// Se o sinal não mudou de estado...
IF bPulse_2s = Special_Variables.Pulse_2s THEN
	// Atualiza temporizador do sinal
	di2sTimer:= di2sTimer + ProjectConstants.iMainTaskInterval;
	// Indica erro caso o sinal não tenha mudado de estado no dobro do tempo esperado
	IF di2sTimer > 2000 THEN bPulse2sFail:= TRUE; END_IF
// Se o sinal mudou de estado...
ELSE
	// Indica erro caso o sinal tenha mudado de estado antes ou depois do tempo esperado
	IF	di2sTimer < (2000 / 2 - diMainTaskIntervalGapMs) OR
		di2sTimer > (2000 / 2 + diMainTaskIntervalGapMs) THEN
			bPulse2sFail:= TRUE;
	END_IF
	// Inicializa o temporizador do sinal
	di2sTimer:= ProjectConstants.iMainTaskInterval;
	// Memoriza o estado atual do sinal
	bPulse_2s:= Special_Variables.Pulse_2s;
END_IF

// Se o sinal não mudou de estado...
IF bPulse_5s = Special_Variables.Pulse_5s THEN
	// Atualiza temporizador do sinal
	di5sTimer:= di5sTimer + ProjectConstants.iMainTaskInterval;
	// Indica erro caso o sinal não tenha mudado de estado no dobro do tempo esperado
	IF di5sTimer > 5000 THEN bPulse5sFail:= TRUE; END_IF
// Se o sinal mudou de estado...
ELSE
	// Indica erro caso o sinal tenha mudado de estado antes ou depois do tempo esperado
	IF	di5sTimer < (5000 / 2 - diMainTaskIntervalGapMs) OR
		di5sTimer > (5000 / 2 + diMainTaskIntervalGapMs) THEN
			bPulse5sFail:= TRUE;
	END_IF
	// Inicializa o temporizador do sinal
	di5sTimer:= ProjectConstants.iMainTaskInterval;
	// Memoriza o estado atual do sinal
	bPulse_5s:= Special_Variables.Pulse_5s;
END_IF

// Se o sinal não mudou de estado...
IF bPulse_10s = Special_Variables.Pulse_10s THEN
	// Atualiza temporizador do sinal
	di10sTimer:= di10sTimer + ProjectConstants.iMainTaskInterval;
	// Indica erro caso o sinal não tenha mudado de estado no dobro do tempo esperado
	IF di10sTimer > 10000 THEN bPulse10sFail:= TRUE; END_IF
// Se o sinal mudou de estado...
ELSE
	// Indica erro caso o sinal tenha mudado de estado antes ou depois do tempo esperado
	IF	di10sTimer < (10000 / 2 - diMainTaskIntervalGapMs) OR
		di10sTimer > (10000 / 2 + diMainTaskIntervalGapMs) THEN
			bPulse10sFail:= TRUE;
	END_IF
	// Inicializa o temporizador do sinal
	di10sTimer:= ProjectConstants.iMainTaskInterval;
	// Memoriza o estado atual do sinal
	bPulse_10s:= Special_Variables.Pulse_10s;
END_IF

// Se o sinal não mudou de estado...
IF bPulse_30s = Special_Variables.Pulse_30s THEN
	// Atualiza temporizador do sinal
	di30sTimer:= di30sTimer + ProjectConstants.iMainTaskInterval;
	// Indica erro caso o sinal não tenha mudado de estado no dobro do tempo esperado
	IF di30sTimer > 30000 THEN bPulse30sFail:= TRUE; END_IF
// Se o sinal mudou de estado...
ELSE
	// Indica erro caso o sinal tenha mudado de estado antes ou depois do tempo esperado
	IF	di30sTimer < (30000 / 2 - diMainTaskIntervalGapMs) OR
		di30sTimer > (30000 / 2 + diMainTaskIntervalGapMs) THEN
			bPulse30sFail:= TRUE;
	END_IF
	// Inicializa o temporizador do sinal
	di30sTimer:= ProjectConstants.iMainTaskInterval;
	// Memoriza o estado atual do sinal
	bPulse_30s:= Special_Variables.Pulse_30s;
END_IF

// Se o sinal não mudou de estado...
IF bPulse_60s = Special_Variables.Pulse_60s THEN
	// Atualiza temporizador do sinal
	di60sTimer:= di60sTimer + ProjectConstants.iMainTaskInterval;
	// Indica erro caso o sinal não tenha mudado de estado no dobro do tempo esperado
	IF di60sTimer > 60000 THEN bPulse60sFail:= TRUE; END_IF
// Se o sinal mudou de estado...
ELSE
	// Indica erro caso o sinal tenha mudado de estado antes ou depois do tempo esperado
	IF	di60sTimer < (60000 / 2 - diMainTaskIntervalGapMs) OR
		di60sTimer > (60000 / 2 + diMainTaskIntervalGapMs) THEN
			bPulse60sFail:= TRUE;
	END_IF
	// Inicializa o temporizador do sinal
	di60sTimer:= ProjectConstants.iMainTaskInterval;
	// Memoriza o estado atual do sinal
	bPulse_60s:= Special_Variables.Pulse_60s;
END_IF

// Realiza as consistências para identificar falhas nos demais sinais da GVL Special_Variables
bPulseScanFail:= bPulseScanFail OR Special_Variables.Pulse_Scan <> bPulse_Scan;
// Consistência em função do retorno da chamada da função
IF udiSystemTimeCall = NextoStandard.RTC_STATUS.NO_ERROR THEN
	// Só consiste se os milisegundos ainda não viraram...
	IF Special_Variables.System_Time.wMilliseconds <= System_Time.wMilliseconds THEN
		bSystemTimeFail:= bSystemTimeFail OR	Special_Variables.System_Time.byDayOfMonth <> System_Time.byDayOfMonth OR
												Special_Variables.System_Time.byHours <> System_Time.byHours OR
												Special_Variables.System_Time.byMinutes <> System_Time.byMinutes OR
												Special_Variables.System_Time.byMonth <> System_Time.byMonth OR
												Special_Variables.System_Time.bySeconds <> System_Time.bySeconds OR
												Special_Variables.System_Time.wYear <> System_Time.wYear;
		bHourMinuteFail:= bHourMinuteFail OR Special_Variables.Hour_Minute <> Hour_Minute;
		bDayOfWeekFail:= bDayOfWeekFail OR Special_Variables.Day_Of_Week <> Day_Of_Week;
	END_IF
ELSE
	// Indica que chamada de função retornou erro
	bSystemTimeCall:= TRUE;
	// Memoriza o erro para fins de depuração
	udiSystemTimeCallErr:= udiSystemTimeCall;
END_IF
bDayOfWeekNull:= bDayOfWeekNull OR Day_Of_Week = NextoStandard.DAYS_OF_WEEK.INVALID_DAY;
bMainTaskFail:= bMainTaskFail OR Special_Variables.udiMainTaskInterval <> DINT_TO_UDINT(ProjectConstants.iMainTaskInterval * 1000);

// Só consiste as variáveis especiais redundantes na UCP ativa, pois na UCP não-ativa elas estão um ciclo atrasadas
IF DG_NX4010.tRedundancy.RedDgnLoc.sGeneral_Diag.eRedState = REDUNDANCY_STATE.ACTIVE THEN
	// Realiza as consitências em relação as variáveis especiais redundantes
	CheckSpecialVarsRed();
END_IF

// Resume as falhas identificadas neste cluster
NonRedPointer.pbSpecialVariablesLoc^:=	bPulse100msFail	OR	CheckSpecialVarsRed.bPulse100msFail OR
										bPulse500msFail OR	CheckSpecialVarsRed.bPulse500msFail OR
										bPulse1sFail	OR	CheckSpecialVarsRed.bPulse1sFail OR
										bPulse2sFail	OR	CheckSpecialVarsRed.bPulse2sFail OR
										bPulse5sFail	OR	CheckSpecialVarsRed.bPulse5sFail OR
										bPulse10sFail	OR	CheckSpecialVarsRed.bPulse10sFail OR
										bPulse30sFail	OR	CheckSpecialVarsRed.bPulse30sFail OR
										bPulse60sFail	OR	CheckSpecialVarsRed.bPulse60sFail OR
										bPulseScanFail	OR	CheckSpecialVarsRed.bPulseScanFail OR
										bSystemTimeCall	OR
										bSystemTimeFail	OR
										bHourMinuteFail	OR
										bDayOfWeekFail	OR
										bDayOfWeekNull	OR
										bMainTaskFail	OR
										FALSE;

// Resume as falhas identificadas em ambos os clusters
PersistentVars.bSpecialVariables:=	PersistentVars.bSpecialVariables OR
									NonRedPointer.pbSpecialVariablesLoc^ OR
									NonRedPointer.pbSpecialVariablesRem^ OR
									FALSE;

// Registra o tempo do sistema
Return_SysTimeGetUs_2:= SysTimeCore.SysTimeGetUs(uliPouEndTime);

// Calcula duração mínima/máxima desta POU
MinMaxTimes.uliPouMinTime_CheckSpecialVars:= MIN(MinMaxTimes.uliPouMinTime_CheckSpecialVars, uliPouEndTime - uliPouIniTime);
MinMaxTimes.uliPouMaxTime_CheckSpecialVars:= MAX(MinMaxTimes.uliPouMaxTime_CheckSpecialVars, uliPouEndTime - uliPouIniTime);

END_PROGRAM

// Device/Application/UserPOUs/NonSkippedPrg
PROGRAM NonSkippedPrg
VAR
	{attribute 'symbol' := 'read'}
	OPCRedundancyActive : BOOL;
	byLocalRedStateOld : REDUNDANCY_STATE;
	uliPouIniTime : ULINT;
	uliPouEndTime : ULINT;
	uliPouAvgTime : ARRAY [1..100] OF ULINT;
	uliPouSumTime : ULINT;
	iPouTimeIndex : INT := 1;
	bFirstCycle : BOOL := 1;
	iIndex : INT;
	tonNetVar : TON;
	tTimeNetVar : TIME := TIME#2S0MS;
	
	udiContadorDeCallBack_Last : UDINT;
	udiContadorDeCallBack_timeout : UDINT;
	udiContadorDeCallBack_timeout_max : UDINT;
		
	{attribute 'symbol' := 'read'}
	DG_NX3030_ACTIVE_tDetailed_Thermometer_diTemperature : DINT;	
	
END_VAR

// Registra o tempo do sistema
SysTimeGetUs(uliPouIniTime);

// Registra a data e hora desta chamada (utilizado em várias POUs)
NextoStandard.GetDateAndTime(NonRedData.xNonSkippedPrgDateAndTime);

// Consistência das variáveis especiais (chamada cíclica)
CheckSpecialVariables();

tonNetVar.PT:=tTimeNetVar;
// Código utilizado na redundância OPC
IF fbRedundancyManagement.m_fbDiagnosticsLocal.eRedState = REDUNDANCY_STATE.ACTIVE THEN
      OPCRedundancyActive := TRUE;
	  tonNetVar();
	  tonNetVar.IN:=TRUE;
	  IF tonNetVar.Q = TRUE THEN
		  NetVar_Application_GVL.TxPDOs_UDP[0].bActive:=TRUE;
		  NetVar_Application_GVL.TxPDOs_UDP[1].bActive:=TRUE;
		  NetVar_Application_GVL.TxPDOs_UDP[2].bActive:=TRUE;
		  NetVar_Application_GVL.TxPDOs_UDP[3].bActive:=TRUE;
		  NetVar_Application_GVL.TxPDOs_UDP[4].bActive:=TRUE;
	  END_IF
ELSE
      OPCRedundancyActive := FALSE;
	  NetVar_Application_GVL.TxPDOs_UDP[0].bActive:=FALSE;
	  NetVar_Application_GVL.TxPDOs_UDP[1].bActive:=FALSE;
	  NetVar_Application_GVL.TxPDOs_UDP[2].bActive:=FALSE;
	  NetVar_Application_GVL.TxPDOs_UDP[3].bActive:=FALSE;
	  NetVar_Application_GVL.TxPDOs_UDP[4].bActive:=FALSE;
	  tonNetVar.IN:=FALSE;
END_IF

// Rotina responsável pela leitura das informações de firmware dos módulos do barramento local
IF DG_NX3030.tSummarized.bAbsentModules <> 0 OR SymbolicsNonRedundant.bReadHWVersions = FALSE THEN
	// Realiza Leitura do FW dos módulos no barramento
	ReadHwVersions();
END_IF
// Rotina que envia as informações de firmware do cluster não ativo para o ativo
WriteHwVersionsNonActive();

// Rotina de salvamento do estado de redundância deste PLC dos ciclos anteriores
NonRedData.aeLastRedState[2]:= NonRedData.aeLastRedState[1];
NonRedData.aeLastRedState[1]:= NonRedData.aeLastRedState[0];
NonRedData.aeLastRedState[0]:= DG_NX4010.tRedundancy.RedDgnLoc.sGeneral_Diag.eRedState;

// MODBUS_Slave_1: copia o valor das saídas para as entradas
ATs.abyModbus1Status:= ATs.abyModbus1Coils;
ATs.awModbus1InputReg:= ATs.awModbus1Holding;

// Comunicação MQTT
IF fbRedundancyManagement.m_fbDiagnosticsLocal.eRedState = REDUNDANCY_STATE.ACTIVE THEN
	MQTT();
END_IF


DG_NX3030_ACTIVE_tDetailed_Thermometer_diTemperature:= DG_NX3030.tDetailed.Thermometer.diTemperature;


// Faz uma copia do pedido de inicio do teste para uso nas demais POUs
Symbolics.bStartTestCopy:= PersistentVars.bStartTest;
// Retorna se o teste estiver desabilitado
IF PersistentVars.bStartTest = FALSE THEN
	RETURN;
END_IF

// Verifica solicitação de reinicialização do super teste
IF PersistentVars.bEnableCleanStats = TRUE THEN
	// Reseta solicitação de reinicialização
	PersistentVars.bEnableCleanStats:= FALSE;
	// Solicita a incialização de todas as variáveis
	CleanStats();
	SymbolicsNonRedundant.bReadHWVersions:= FALSE;
	SymbolicsNonRedundant.bEnableCleanStats_CheckForcing:= TRUE;
	SymbolicsNonRedundant.bEnableCleanStats_CheckRam:= TRUE;
	SymbolicsNonRedundant.bEnableCleanStats_CheckSntp:= TRUE;
	SymbolicsNonRedundant.bEnableCleanStats_CheckRedData:= TRUE;
	Symbolics.bEnableCleanStats_ActivePrg:= TRUE;
	Symbolics.bEnableCleanStats_CheckNVL:= TRUE;
	SymbolicsNonRedundant.bEnableCleanStats_NonSkippedPrg:= TRUE;
	SymbolicsNonRedundant.bEnableCleanStats_CheckDiagsRetain:= TRUE;
END_IF


CycleTimes();			// Registra os tempos de ciclo máximo, mínimo e médio das tarefas
CheckModbus1();			// Consistência dos objetos de comunicação MODBUS Serial
CheckRedData();			// Consistência dos dados redundantes
CheckSntp();			// Consistência da atualização do relógio via SNTP
UserLog();				// Consistência e geração do LOG de usuário
CheckForcing();			// Consistência dos forçamentos
CheckDiagsRetain();		// Consistência e resumo dos diagnósticos ativos
CheckRam();				// Consistência da memória RAM da UCP	
//DaylightSavingTime();	// Ajuste do timezone em função do horário de verão

// Reseta a indicação de alteração de estado de redundância deste PLC
NonRedData.bRedStateChanged:= FALSE;
// Detecta alteração no estado de redundância deste PLC
IF DG_NX4010.tRedundancy.RedDgnLoc.sGeneral_Diag.eRedState <> byLocalRedStateOld THEN
	// Salva o estado de redundância atual deste PLC
	byLocalRedStateOld:= DG_NX4010.tRedundancy.RedDgnLoc.sGeneral_Diag.eRedState;
	// Indica que o estado de redundância deste PLC alterou
	NonRedData.bRedStateChanged:= TRUE;
	// Se este PLC é o ativo...
	IF DG_NX4010.tRedundancy.RedDgnLoc.sGeneral_Diag.eRedState = REDUNDANCY_STATE.ACTIVE THEN
		// Habilita os MODBUS Ethernet clientes 
		System_Diagnostics.DG_MODBUS_Client_2.tCommand.bRestart:= TRUE;
		System_Diagnostics.DG_MODBUS_Client_3.tCommand.bRestart:= TRUE;
		System_Diagnostics.DG_MODBUS_Client_4.tCommand.bRestart:= TRUE;
	// Se este PLC é não-ativo...
	ELSE
		// Desabilita os MODBUS Ethernet clientes
		System_Diagnostics.DG_MODBUS_Client_2.tCommand.bStop:= TRUE;
		System_Diagnostics.DG_MODBUS_Client_3.tCommand.bStop:= TRUE;
		System_Diagnostics.DG_MODBUS_Client_4.tCommand.bStop:= TRUE;
		// Inicializa temporizador para atrasar a consistência dos valores lidos,
		// pois quando o PLC irá assumir como ativo, vai levar alguns ciclos até
		// que a comunicação MODBUS/Profibus seja estabelecida e estabilizada
		NonRedData.iProfibus5DigTimer:= - ProjectConstants.iTimeToSkipAsActive;
		NonRedData.iProfibus10AnaTimer:= - ProjectConstants.iTimeToSkipAsActive;
		NonRedData.iProfibus3DigTimer:= - ProjectConstants.iTimeToSkipAsActive;
		NonRedData.iProfibus98DigTimer:= - ProjectConstants.iTimeToSkipAsActive;
		NonRedData.iProfibus99DigTimer:= - ProjectConstants.iTimeToSkipAsActive;
		NonRedData.iProfibus99Dig1005Timer:= - ProjectConstants.iTimeToSkipAsActive;
		NonRedData.iProfibusNXTimer:= - ProjectConstants.iTimeToSkipAsActive;
		NonRedData.iProfibus99AnaTimer:= - ProjectConstants.iTimeToSkipAsActive;
		// Indicador de necessidade de inicializar as variáveis de geração de SOE
		// a partir dos diagnósticos retentivos
		NonRedData.bSoeFirstCheckCycle:= TRUE;
	END_IF
END_IF



/// Depuração do BUG 19183
IF SymbolicsNonRedundant.bEnableCleanStats_NonSkippedPrg THEN
	// Reseta os contadores de sobra de timeout da sincronismo
	FOR iIndex:= 0 TO 99 DO
		MinMaxTimes.auliRedRemainTimeoutCounter[iIndex]:= 0;
	END_FOR
	// Modifica o timeout de redundancia original (que era 111)
	redundancy_time_values.g_dwRedundancyTimeout_ms:= 151;
	SymbolicsNonRedundant.bEnableCleanStats_NonSkippedPrg:= FALSE;
ELSIF redundancy_time_values.g_uiLastTimeout <= 99 THEN
	// Incrementa a variável que conta o número de vezes que sobrou o respectivo tempo de sincronismo (índice) 
	MinMaxTimes.auliRedRemainTimeoutCounter[redundancy_time_values.g_uiLastTimeout]:= MinMaxTimes.auliRedRemainTimeoutCounter[redundancy_time_values.g_uiLastTimeout] + 1;
END_IF

//################################################################################################################


// Devido a 3S ter alterado o funcionamento do vfInit sem a Altus saber,
// o funcionamento da sincronização de ponteiros da redundância foi afetada.
// Essa variável interna "Callback_vfInit_Counter" sempre deve ser incrementada
// caso pare de incrementar, significa que a redundância pode apresentar problemas
// na sincronização dos dados.

IF fbRedundancyManagement.m_fbDiagnosticsLocal.eRedState = REDUNDANCY_STATE.STANDBY THEN
	// Confere se o valor mudou de um ciclo para outro
	IF Callback_vfInit_Counter <> udiContadorDeCallBack_Last THEN	
		udiContadorDeCallBack_Last:= Callback_vfInit_Counter;
		udiContadorDeCallBack_timeout:=0;
	ELSE
		udiContadorDeCallBack_timeout:= udiContadorDeCallBack_timeout+1;
	END_IF
	udiContadorDeCallBack_timeout_max:=MAX(udiContadorDeCallBack_timeout_max, udiContadorDeCallBack_timeout);
	// Todos os testes exeutados até agora, o valor máximo registrado foi 1.
	IF udiContadorDeCallBack_timeout_max > 1 THEN
		PersistentVars.iSyncFailCallback_vfInit:= PersistentVars.iSyncFailCallback_vfInit+1;
	END_IF
END_IF


//Esse hotfix deve ser usado quando em versões 3.11 a 3.13.
(* hotfix para versão 3.11 a 3.13 *)
 //  {implicit on}	
//   Callback_vfInit(0);
//   {implicit off}
//################################################################################################################



// Registra o tempo do sistema
SysTimeGetUs(uliPouEndTime);

// Calcula duração média desta POU
uliPouSumTime:= uliPouSumTime - uliPouAvgTime[iPouTimeIndex];
uliPouAvgTime[iPouTimeIndex]:= uliPouEndTime - uliPouIniTime;
uliPouSumTime:= uliPouSumTime + uliPouAvgTime[iPouTimeIndex];
// Calcula duração mínima/média/máxima desta POU
MinMaxTimes.uliPouMinTime_NonSkippedPrg:= MIN(MinMaxTimes.uliPouMinTime_NonSkippedPrg, uliPouAvgTime[iPouTimeIndex]);
MinMaxTimes.uliPouAvgTime_NonSkippedPrg:= uliPouSumTime/(SIZEOF(uliPouAvgTime)/SIZEOF(uliPouAvgTime[1]));
MinMaxTimes.uliPouMaxTime_NonSkippedPrg:= MAX(MinMaxTimes.uliPouMaxTime_NonSkippedPrg, uliPouAvgTime[iPouTimeIndex]);
// Proximo indice para cálculo da duração média desta POU
iPouTimeIndex:= iPouTimeIndex + 1;
IF iPouTimeIndex > ULINT_TO_INT(SIZEOF(uliPouAvgTime)/SIZEOF(uliPouAvgTime[1])) THEN
	iPouTimeIndex:= 1;
END_IF

END_PROGRAM

// Device/Application/UserPOUs/Non-Redundant/ReadHwVersions
PROGRAM ReadHwVersions
VAR
	pSlave : POINTER TO NextoSlave;
	dwRevisionID : ARRAY [0..31] OF DWORD;
	uiAddress : ARRAY [0..31] OF UINT;
	dwProductID : ARRAY [0..31] OF DWORD;
	byIndex : BYTE;
	iIndex : INT;
END_VAR

//*****************************************************************************
// Autor(es): Roberto Martiny
// Descrição:
// Esta POU realiza a leitura do firmware via NextoBus e armazena as informações para serem lidas via SCADA.
//*****************************************************************************

IF DG_NX4010.tRedundancy.RedDgnLoc.sGeneral_Diag.ePLC_ID = CLUCONF_ID.PLC_A THEN
	// Realiza a leitura do firmware via NextoBus. 
			IF g_pFirstMaster <> 0 THEN
			pSlave := g_pFirstMaster^.FirstSlave;
			///pSlave := Configuration.FirstSlave;
			WHILE pSlave <> 0 DO
			   dwRevisionID[byIndex] := pSlave^.RevisionID; // Leitura da versão fo firmware.
			   uiAddress[byIndex] := pSlave^.PhysSlaveAddr; // Leitura do rack e slot.
			   dwProductID[byIndex] := pSlave^.ProductID; // Leitura do tipo do produto.
			   byIndex:=byIndex+1;
			   pSlave := pSlave^.NextInstance;
			END_WHILE
			END_IF
		byIndex:= 0;
		
		FOR iIndex:=0 TO 31 DO
		// Consulta Informações Rack 00 Slot 04
			IF uiAddress[iIndex] = 16#0004 THEN
				HwVersions.eR00S04_NX4010_PlcA.iIndex:= iIndex;
			END_IF
			HwVersions.eR00S04_NX4010_PlcA.dwFirmwareVersion:= DwRevisionID[HwVersions.eR00S04_NX4010_PlcA.iIndex];
			HwVersions.eR00S04_NX4010_PlcA.dwProductID:= DwProductID[HwVersions.eR00S04_NX4010_PlcA.iIndex];
			HwVersions.eR00S04_NX4010_PlcA.uiSlaveAddress:= uiAddress[HwVersions.eR00S04_NX4010_PlcA.iIndex];
			
		// Consulta Informações Rack 00 Slot 06
			IF uiAddress[iIndex] = 16#0006 THEN
				HwVersions.eR00S06_NX5001_PlcA.iIndex:= iIndex;
			END_IF
			HwVersions.eR00S06_NX5001_PlcA.dwFirmwareVersion:= DwRevisionID[HwVersions.eR00S06_NX5001_PlcA.iIndex];
			HwVersions.eR00S06_NX5001_PlcA.dwProductID:= DwProductID[HwVersions.eR00S06_NX5001_PlcA.iIndex];
			HwVersions.eR00S06_NX5001_PlcA.uiSlaveAddress:= uiAddress[HwVersions.eR00S06_NX5001_PlcA.iIndex];	
			
		// Consulta Informações Rack 00 Slot 08
			IF uiAddress[iIndex] = 16#0008 THEN
				HwVersions.eR00S08_NX5001_PlcA.iIndex:= iIndex;
			END_IF
			HwVersions.eR00S08_NX5001_PlcA.dwFirmwareVersion:= DwRevisionID[HwVersions.eR00S08_NX5001_PlcA.iIndex];
			HwVersions.eR00S08_NX5001_PlcA.dwProductID:= DwProductID[HwVersions.eR00S08_NX5001_PlcA.iIndex];
			HwVersions.eR00S08_NX5001_PlcA.uiSlaveAddress:= uiAddress[HwVersions.eR00S08_NX5001_PlcA.iIndex];
	
		// Consulta Informações Rack 00 Slot 10
			IF uiAddress[iIndex] = 16#000A THEN
				HwVersions.eR00S10_NX5000_PlcA.iIndex:= iIndex;
			END_IF
			HwVersions.eR00S10_NX5000_PlcA.dwFirmwareVersion:= DwRevisionID[HwVersions.eR00S10_NX5000_PlcA.iIndex];
			HwVersions.eR00S10_NX5000_PlcA.dwProductID:= DwProductID[HwVersions.eR00S10_NX5000_PlcA.iIndex];
			HwVersions.eR00S10_NX5000_PlcA.uiSlaveAddress:= uiAddress[HwVersions.eR00S10_NX5000_PlcA.iIndex];
	
		// Consulta Informações Rack 00 Slot 12
			IF uiAddress[iIndex] = 16#000C THEN
				HwVersions.eR00S12_NX5000_PlcA.iIndex:= iIndex;
			END_IF
			HwVersions.eR00S12_NX5000_PlcA.dwFirmwareVersion:= DwRevisionID[HwVersions.eR00S12_NX5000_PlcA.iIndex];
			HwVersions.eR00S12_NX5000_PlcA.dwProductID:= DwProductID[HwVersions.eR00S12_NX5000_PlcA.iIndex];
			HwVersions.eR00S12_NX5000_PlcA.uiSlaveAddress:= uiAddress[HwVersions.eR00S12_NX5000_PlcA.iIndex];
			
		// Consulta Informações Rack 00 Slot 16
			IF uiAddress[iIndex] = 16#0010 THEN
				HwVersions.eR00S16_NX5001_PlcA.iIndex:= iIndex;
			END_IF
			HwVersions.eR00S16_NX5001_PlcA.dwFirmwareVersion:= DwRevisionID[HwVersions.eR00S16_NX5001_PlcA.iIndex];
			HwVersions.eR00S16_NX5001_PlcA.dwProductID:= DwProductID[HwVersions.eR00S16_NX5001_PlcA.iIndex];
			HwVersions.eR00S16_NX5001_PlcA.uiSlaveAddress:= uiAddress[HwVersions.eR00S16_NX5001_PlcA.iIndex];	
			
		// Consulta Informações Rack 00 Slot 20
			IF uiAddress[iIndex] = 16#0014 THEN
				HwVersions.eR00S20_NX5000_PlcA.iIndex:= iIndex;
			END_IF
			HwVersions.eR00S20_NX5000_PlcA.dwFirmwareVersion:= DwRevisionID[HwVersions.eR00S20_NX5000_PlcA.iIndex];
			HwVersions.eR00S20_NX5000_PlcA.dwProductID:= DwProductID[HwVersions.eR00S20_NX5000_PlcA.iIndex];
			HwVersions.eR00S20_NX5000_PlcA.uiSlaveAddress:= uiAddress[HwVersions.eR00S20_NX5000_PlcA.iIndex];			
		END_FOR	
	
		HwVersions.eR00S02_NX3030_PlcA.abyBootloaderVersion[0]:= DG_NX3030.tDetailed.Target.abyBootloaderVersion[0];
		HwVersions.eR00S02_NX3030_PlcA.abyBootloaderVersion[1]:= DG_NX3030.tDetailed.Target.abyBootloaderVersion[1];
		HwVersions.eR00S02_NX3030_PlcA.abyBootloaderVersion[2]:= DG_NX3030.tDetailed.Target.abyBootloaderVersion[2];
		HwVersions.eR00S02_NX3030_PlcA.abyBootloaderVersion[3]:= DG_NX3030.tDetailed.Target.abyBootloaderVersion[3];
		HwVersions.eR00S02_NX3030_PlcA.abyCPUVersion[0]:= DG_NX3030.tDetailed.Target.abyCPUVersion[0];
		HwVersions.eR00S02_NX3030_PlcA.abyCPUVersion[1]:= DG_NX3030.tDetailed.Target.abyCPUVersion[1];
		HwVersions.eR00S02_NX3030_PlcA.abyCPUVersion[2]:= DG_NX3030.tDetailed.Target.abyCPUVersion[2];
		HwVersions.eR00S02_NX3030_PlcA.abyCPUVersion[3]:= DG_NX3030.tDetailed.Target.abyCPUVersion[3];
		HwVersions.eR00S02_NX3030_PlcA.abyProcAuxVersion[0] := DG_NX3030.tDetailed.Target.abyAuxprocVersion[0];
		HwVersions.eR00S02_NX3030_PlcA.abyProcAuxVersion[1] := DG_NX3030.tDetailed.Target.abyAuxprocVersion[1];
		HwVersions.eR00S02_NX3030_PlcA.abyProcAuxVersion[2] := DG_NX3030.tDetailed.Target.abyAuxprocVersion[2];
		HwVersions.eR00S02_NX3030_PlcA.abyProcAuxVersion[3] := DG_NX3030.tDetailed.Target.abyAuxprocVersion[3];
		HwVersions.eR00S02_NX3030_PlcA.dwCPUModel:= DG_NX3030.tDetailed.Target.dwCPUModel;	
		
		SymbolicsNonRedundant.bReadHWVersions:= TRUE;
END_IF

IF DG_NX4010.tRedundancy.RedDgnLoc.sGeneral_Diag.ePLC_ID = CLUCONF_ID.PLC_B THEN
	// Realiza a leitura do firmware via NextoBus. 
			IF g_pFirstMaster <> 0 THEN
			pSlave := g_pFirstMaster^.FirstSlave;
			WHILE pSlave <> 0 DO
			   dwRevisionID[byIndex] := pSlave^.RevisionID; // Leitura da versão fo firmware.
			   uiAddress[byIndex] := pSlave^.PhysSlaveAddr; // Leitura do rack e slot.
			   dwProductID[byIndex] := pSlave^.ProductID; // Leitura do tipo do produto.
			   byIndex:=byIndex+1;
			   pSlave := pSlave^.NextInstance;
			END_WHILE
		byIndex:= 0;
		END_IF
		FOR iIndex:=0 TO 31 DO
			// Consulta Informações Rack 00 Slot 04
			IF uiAddress[iIndex] = 16#0004 THEN
				HwVersions.eR00S04_NX4010_PlcB.iIndex:= iIndex;
			END_IF
			HwVersions.eR00S04_NX4010_PlcB.dwFirmwareVersion:= DwRevisionID[HwVersions.eR00S04_NX4010_PlcB.iIndex];
			HwVersions.eR00S04_NX4010_PlcB.dwProductID:= DwProductID[HwVersions.eR00S04_NX4010_PlcB.iIndex];
			HwVersions.eR00S04_NX4010_PlcB.uiSlaveAddress:= uiAddress[HwVersions.eR00S04_NX4010_PlcB.iIndex];
			
		// Consulta Informações Rack 00 Slot 06
			IF uiAddress[iIndex] = 16#0006 THEN
				HwVersions.eR00S06_NX5001_PlcB.iIndex:= iIndex;
			END_IF
			HwVersions.eR00S06_NX5001_PlcB.dwFirmwareVersion:= DwRevisionID[HwVersions.eR00S06_NX5001_PlcB.iIndex];
			HwVersions.eR00S06_NX5001_PlcB.dwProductID:= DwProductID[HwVersions.eR00S06_NX5001_PlcB.iIndex];
			HwVersions.eR00S06_NX5001_PlcB.uiSlaveAddress:= uiAddress[HwVersions.eR00S06_NX5001_PlcB.iIndex];	
			
		// Consulta Informações Rack 00 Slot 08
			IF uiAddress[iIndex] = 16#0008 THEN
				HwVersions.eR00S08_NX5001_PlcB.iIndex:= iIndex;
			END_IF
			HwVersions.eR00S08_NX5001_PlcB.dwFirmwareVersion:= DwRevisionID[HwVersions.eR00S08_NX5001_PlcB.iIndex];
			HwVersions.eR00S08_NX5001_PlcB.dwProductID:= DwProductID[HwVersions.eR00S08_NX5001_PlcB.iIndex];
			HwVersions.eR00S08_NX5001_PlcB.uiSlaveAddress:= uiAddress[HwVersions.eR00S08_NX5001_PlcB.iIndex];
	
		// Consulta Informações Rack 00 Slot 10
			IF uiAddress[iIndex] = 16#000A THEN
				HwVersions.eR00S10_NX5000_PlcB.iIndex:= iIndex;
			END_IF
			HwVersions.eR00S10_NX5000_PlcB.dwFirmwareVersion:= DwRevisionID[HwVersions.eR00S10_NX5000_PlcB.iIndex];
			HwVersions.eR00S10_NX5000_PlcB.dwProductID:= DwProductID[HwVersions.eR00S10_NX5000_PlcB.iIndex];
			HwVersions.eR00S10_NX5000_PlcB.uiSlaveAddress:= uiAddress[HwVersions.eR00S10_NX5000_PlcB.iIndex];
	
		// Consulta Informações Rack 00 Slot 12
			IF uiAddress[iIndex] = 16#000C THEN
				HwVersions.eR00S12_NX5000_PlcB.iIndex:= iIndex;
			END_IF
			HwVersions.eR00S12_NX5000_PlcB.dwFirmwareVersion:= DwRevisionID[HwVersions.eR00S12_NX5000_PlcB.iIndex];
			HwVersions.eR00S12_NX5000_PlcB.dwProductID:= DwProductID[HwVersions.eR00S12_NX5000_PlcB.iIndex];
			HwVersions.eR00S12_NX5000_PlcB.uiSlaveAddress:= uiAddress[HwVersions.eR00S12_NX5000_PlcB.iIndex];
			
		// Consulta Informações Rack 00 Slot 16
			IF uiAddress[iIndex] = 16#0010 THEN
				HwVersions.eR00S16_NX5001_PlcB.iIndex:= iIndex;
			END_IF
			HwVersions.eR00S16_NX5001_PlcB.dwFirmwareVersion:= DwRevisionID[HwVersions.eR00S16_NX5001_PlcB.iIndex];
			HwVersions.eR00S16_NX5001_PlcB.dwProductID:= DwProductID[HwVersions.eR00S16_NX5001_PlcB.iIndex];
			HwVersions.eR00S16_NX5001_PlcB.uiSlaveAddress:= uiAddress[HwVersions.eR00S16_NX5001_PlcB.iIndex];	
			
		// Consulta Informações Rack 00 Slot 20
			IF uiAddress[iIndex] = 16#0014 THEN
				HwVersions.eR00S20_NX5000_PlcB.iIndex:= iIndex;
			END_IF
			HwVersions.eR00S20_NX5000_PlcB.dwFirmwareVersion:= DwRevisionID[HwVersions.eR00S20_NX5000_PlcB.iIndex];
			HwVersions.eR00S20_NX5000_PlcB.dwProductID:= DwProductID[HwVersions.eR00S20_NX5000_PlcB.iIndex];
			HwVersions.eR00S20_NX5000_PlcB.uiSlaveAddress:= uiAddress[HwVersions.eR00S20_NX5000_PlcB.iIndex];			
		END_FOR	
	
		HwVersions.eR00S02_NX3030_PlcB.abyBootloaderVersion[0]:= DG_NX3030.tDetailed.Target.abyBootloaderVersion[0];
		HwVersions.eR00S02_NX3030_PlcB.abyBootloaderVersion[1]:= DG_NX3030.tDetailed.Target.abyBootloaderVersion[1];
		HwVersions.eR00S02_NX3030_PlcB.abyBootloaderVersion[2]:= DG_NX3030.tDetailed.Target.abyBootloaderVersion[2];
		HwVersions.eR00S02_NX3030_PlcB.abyBootloaderVersion[3]:= DG_NX3030.tDetailed.Target.abyBootloaderVersion[3];
		HwVersions.eR00S02_NX3030_PlcB.abyCPUVersion[0]:= DG_NX3030.tDetailed.Target.abyCPUVersion[0];
		HwVersions.eR00S02_NX3030_PlcB.abyCPUVersion[1]:= DG_NX3030.tDetailed.Target.abyCPUVersion[1];
		HwVersions.eR00S02_NX3030_PlcB.abyCPUVersion[2]:= DG_NX3030.tDetailed.Target.abyCPUVersion[2];
		HwVersions.eR00S02_NX3030_PlcB.abyCPUVersion[3]:= DG_NX3030.tDetailed.Target.abyCPUVersion[3];
		HwVersions.eR00S02_NX3030_PlcB.abyProcAuxVersion[0] := DG_NX3030.tDetailed.Target.abyAuxprocVersion[0];
		HwVersions.eR00S02_NX3030_PlcB.abyProcAuxVersion[1] := DG_NX3030.tDetailed.Target.abyAuxprocVersion[1];
		HwVersions.eR00S02_NX3030_PlcB.abyProcAuxVersion[2] := DG_NX3030.tDetailed.Target.abyAuxprocVersion[2];
		HwVersions.eR00S02_NX3030_PlcB.abyProcAuxVersion[3] := DG_NX3030.tDetailed.Target.abyAuxprocVersion[3];
		HwVersions.eR00S02_NX3030_PlcB.dwCPUModel:= DG_NX3030.tDetailed.Target.dwCPUModel;
		
		SymbolicsNonRedundant.bReadHWVersions:= TRUE;
END_IF

END_PROGRAM

// Device/Application/UserPOUs/Non-Redundant/WriteHwVersionsNonActive
PROGRAM WriteHwVersionsNonActive
VAR
	pSlave : POINTER TO NextoSlave;
	dwRevisionID : ARRAY [0..31] OF DWORD;
	uiAddress : ARRAY [0..31] OF UINT;
	dwProductID : ARRAY [0..31] OF DWORD;
	byIndex : BYTE;
	iIndex : INT;
	uliPouIniTime : ULINT;
	uliPouEndTime : ULINT;
END_VAR

//*****************************************************************************
// Autor(es): Jenifer Dal Magro
// Descrição:
// Esta POU envia as versões de Hardware do PLC não Ativo para o Ativo.
//*****************************************************************************
// Registra o tempo do sistema
SysTimeGetUs(uliPouIniTime);

IF DG_NX4010.tRedundancy.RedDgnLoc.sGeneral_Diag.ePLC_ID = CLUCONF_ID.PLC_A THEN
	IF DG_NX4010.tRedundancy.RedDgnLoc.sGeneral_Diag.eRedState = REDUNDANCY_STATE.ACTIVE THEN
		// Copia as versões de Hardware do PLC B não ativo para suas posições na GVL HwVersions
		// Firmware da CPU
		HwVersions.eR00S02_NX3030_PlcB.abyCPUVersion[0]	:=	DG_NX4010.tRedundancy.RedUsrRem.abyUser[1]	;
		HwVersions.eR00S02_NX3030_PlcB.abyCPUVersion[1]	:=	DG_NX4010.tRedundancy.RedUsrRem.abyUser[2]	;
		HwVersions.eR00S02_NX3030_PlcB.abyCPUVersion[2]	:=	DG_NX4010.tRedundancy.RedUsrRem.abyUser[3]	;
		HwVersions.eR00S02_NX3030_PlcB.abyCPUVersion[3]	:=	DG_NX4010.tRedundancy.RedUsrRem.abyUser[4]	;
		// Bootloader
		HwVersions.eR00S02_NX3030_PlcB.abyBootloaderVersion[0]	:=	DG_NX4010.tRedundancy.RedUsrRem.abyUser[5]	;
		HwVersions.eR00S02_NX3030_PlcB.abyBootloaderVersion[1]	:=	DG_NX4010.tRedundancy.RedUsrRem.abyUser[6]	;
		HwVersions.eR00S02_NX3030_PlcB.abyBootloaderVersion[2]	:=	DG_NX4010.tRedundancy.RedUsrRem.abyUser[7]	;
		HwVersions.eR00S02_NX3030_PlcB.abyBootloaderVersion[3]	:=	DG_NX4010.tRedundancy.RedUsrRem.abyUser[8]	;
		// Pocessador Auxiliar
		HwVersions.eR00S02_NX3030_PlcB.abyProcAuxVersion[0]	:=	DG_NX4010.tRedundancy.RedUsrRem.abyUser[9]	;
		HwVersions.eR00S02_NX3030_PlcB.abyProcAuxVersion[1]	:=	DG_NX4010.tRedundancy.RedUsrRem.abyUser[10]	;
		HwVersions.eR00S02_NX3030_PlcB.abyProcAuxVersion[2]	:=	DG_NX4010.tRedundancy.RedUsrRem.abyUser[11]	;
		HwVersions.eR00S02_NX3030_PlcB.abyProcAuxVersion[3]	:=	DG_NX4010.tRedundancy.RedUsrRem.abyUser[12]	;	
		// Modelo CPU				
		HwVersions.eR00S02_NX3030_PlcB.dwCPUModel			:=	NonRedPointer.pdw02CPUModelRedUsrRem^	;
		// NX4010				
		HwVersions.eR00S04_NX4010_PlcB.dwFirmwareVersion	:=	NonRedPointer.pdw04NX4010FWRedUsrRem^	;
		HwVersions.eR00S04_NX4010_PlcB.dwProductID			:=	NonRedPointer.pdw04NX4010HWRedUsrRem^	;
		// NX50001				
		HwVersions.eR00S06_NX5001_PlcB.dwFirmwareVersion	:=	NonRedPointer.pdw06NX5001FWRedUsrRem^	;
		HwVersions.eR00S06_NX5001_PlcB.dwProductID			:=	NonRedPointer.pdw06NX5001HWRedUsrRem^	;
		HwVersions.eR00S08_NX5001_PlcB.dwFirmwareVersion	:=	NonRedPointer.pdw08NX5001FWRedUsrRem^	;
		HwVersions.eR00S08_NX5001_PlcB.dwProductID			:=	NonRedPointer.pdw08NX5001HWRedUsrRem^	;
		HwVersions.eR00S16_NX5001_PlcB.dwFirmwareVersion	:=	NonRedPointer.pdw16NX5001FWRedUsrRem^	;
		HwVersions.eR00S16_NX5001_PlcB.dwProductID			:=	NonRedPointer.pdw16NX5001HWRedUsrRem^	;
		// NX5000				
		HwVersions.eR00S10_NX5000_PlcB.dwFirmwareVersion	:=	NonRedPointer.pdw10NX5000FWRedUsrRem^	;
		HwVersions.eR00S10_NX5000_PlcB.dwProductID			:=	NonRedPointer.pdw10NX5000HWRedUsrRem^	;
		HwVersions.eR00S12_NX5000_PlcB.dwFirmwareVersion	:=	NonRedPointer.pdw12NX5000FWRedUsrRem^	;
		HwVersions.eR00S12_NX5000_PlcB.dwProductID			:=	NonRedPointer.pdw12NX5000HWRedUsrRem^	;
		HwVersions.eR00S20_NX5000_PlcB.dwFirmwareVersion	:=	NonRedPointer.pdw20NX5000FWRedUsrRem^	;
		HwVersions.eR00S20_NX5000_PlcB.dwProductID			:=	NonRedPointer.pdw20NX5000HWRedUsrRem^	;

		
	ELSIF	DG_NX4010.tRedundancy.RedDgnLoc.sGeneral_Diag.eRedState = REDUNDANCY_STATE.STANDBY	OR
			DG_NX4010.tRedundancy.RedDgnLoc.sGeneral_Diag.eRedState = REDUNDANCY_STATE.INACTIVE	THEN
		// Copia os dados deste PLC para a área de usuário do PLC remoto			
		// Firmware da CPU
		DG_NX4010.tRedundancy.RedUsrLoc.abyUser[1]	:=	HwVersions.eR00S02_NX3030_PlcA.abyCPUVersion[0]	;
		DG_NX4010.tRedundancy.RedUsrLoc.abyUser[2]	:=	HwVersions.eR00S02_NX3030_PlcA.abyCPUVersion[1]	;
		DG_NX4010.tRedundancy.RedUsrLoc.abyUser[3]	:=	HwVersions.eR00S02_NX3030_PlcA.abyCPUVersion[2]	;
		DG_NX4010.tRedundancy.RedUsrLoc.abyUser[4]	:=	HwVersions.eR00S02_NX3030_PlcA.abyCPUVersion[3]	;
		// Bootloader
		DG_NX4010.tRedundancy.RedUsrLoc.abyUser[5]	:=	HwVersions.eR00S02_NX3030_PlcA.abyBootloaderVersion[0]	;
		DG_NX4010.tRedundancy.RedUsrLoc.abyUser[6]	:=	HwVersions.eR00S02_NX3030_PlcA.abyBootloaderVersion[1]	;
		DG_NX4010.tRedundancy.RedUsrLoc.abyUser[7]	:=	HwVersions.eR00S02_NX3030_PlcA.abyBootloaderVersion[2]	;
		DG_NX4010.tRedundancy.RedUsrLoc.abyUser[8]	:=	HwVersions.eR00S02_NX3030_PlcA.abyBootloaderVersion[3]	;
		// Pocessador Auxiliar
		DG_NX4010.tRedundancy.RedUsrLoc.abyUser[9]	:=	HwVersions.eR00S02_NX3030_PlcA.abyProcAuxVersion[0]	;
		DG_NX4010.tRedundancy.RedUsrLoc.abyUser[10]	:=	HwVersions.eR00S02_NX3030_PlcA.abyProcAuxVersion[1]	;
		DG_NX4010.tRedundancy.RedUsrLoc.abyUser[11]	:=	HwVersions.eR00S02_NX3030_PlcA.abyProcAuxVersion[2]	;
		DG_NX4010.tRedundancy.RedUsrLoc.abyUser[12]	:=	HwVersions.eR00S02_NX3030_PlcA.abyProcAuxVersion[3]	;
		// Modelo CPU
		NonRedPointer.pdw02CPUModelRedUsrLoc^	:=	HwVersions.eR00S02_NX3030_PlcA.dwCPUModel	;
		// NX4010
		NonRedPointer.pdw04NX4010FWRedUsrLoc^	:=	HwVersions.eR00S04_NX4010_PlcA.dwFirmwareVersion	;
		NonRedPointer.pdw04NX4010HWRedUsrLoc^	:=	HwVersions.eR00S04_NX4010_PlcA.dwProductID	;
		// NX50001
		NonRedPointer.pdw06NX5001FWRedUsrLoc^	:=	HwVersions.eR00S06_NX5001_PlcA.dwFirmwareVersion	;
		NonRedPointer.pdw06NX5001HWRedUsrLoc^	:=	HwVersions.eR00S06_NX5001_PlcA.dwProductID	;
		NonRedPointer.pdw08NX5001FWRedUsrLoc^	:=	HwVersions.eR00S08_NX5001_PlcA.dwFirmwareVersion	;
		NonRedPointer.pdw08NX5001HWRedUsrLoc^	:=	HwVersions.eR00S08_NX5001_PlcA.dwProductID	;
		NonRedPointer.pdw16NX5001FWRedUsrLoc^	:=	HwVersions.eR00S16_NX5001_PlcA.dwFirmwareVersion	;
		NonRedPointer.pdw16NX5001HWRedUsrLoc^	:=	HwVersions.eR00S16_NX5001_PlcA.dwProductID	;
		// NX5000
		NonRedPointer.pdw10NX5000FWRedUsrLoc^	:=	HwVersions.eR00S10_NX5000_PlcA.dwFirmwareVersion	;
		NonRedPointer.pdw10NX5000HWRedUsrLoc^	:=	HwVersions.eR00S10_NX5000_PlcA.dwProductID	;
		NonRedPointer.pdw12NX5000FWRedUsrLoc^	:=	HwVersions.eR00S12_NX5000_PlcA.dwFirmwareVersion	;
		NonRedPointer.pdw12NX5000HWRedUsrLoc^	:=	HwVersions.eR00S12_NX5000_PlcA.dwProductID	;
		NonRedPointer.pdw20NX5000FWRedUsrLoc^	:=	HwVersions.eR00S20_NX5000_PlcA.dwFirmwareVersion	;
		NonRedPointer.pdw20NX5000HWRedUsrLoc^	:=	HwVersions.eR00S20_NX5000_PlcA.dwProductID	;

			
			
	END_IF
END_IF

IF DG_NX4010.tRedundancy.RedDgnLoc.sGeneral_Diag.ePLC_ID = CLUCONF_ID.PLC_B THEN
	IF DG_NX4010.tRedundancy.RedDgnLoc.sGeneral_Diag.eRedState = REDUNDANCY_STATE.ACTIVE THEN
		// Copia as versões de Hardware do PLC A não ativo para suas posições na GVL HwVersions
		// Firmware da CPU
		HwVersions.eR00S02_NX3030_PlcA.abyCPUVersion[0]	:=	DG_NX4010.tRedundancy.RedUsrRem.abyUser[1]	;
		HwVersions.eR00S02_NX3030_PlcA.abyCPUVersion[1]	:=	DG_NX4010.tRedundancy.RedUsrRem.abyUser[2]	;
		HwVersions.eR00S02_NX3030_PlcA.abyCPUVersion[2]	:=	DG_NX4010.tRedundancy.RedUsrRem.abyUser[3]	;
		HwVersions.eR00S02_NX3030_PlcA.abyCPUVersion[3]	:=	DG_NX4010.tRedundancy.RedUsrRem.abyUser[4]	;
		// Bootloader
		HwVersions.eR00S02_NX3030_PlcA.abyBootloaderVersion[0]	:=	DG_NX4010.tRedundancy.RedUsrRem.abyUser[5]	;
		HwVersions.eR00S02_NX3030_PlcA.abyBootloaderVersion[1]	:=	DG_NX4010.tRedundancy.RedUsrRem.abyUser[6]	;
		HwVersions.eR00S02_NX3030_PlcA.abyBootloaderVersion[2]	:=	DG_NX4010.tRedundancy.RedUsrRem.abyUser[7]	;
		HwVersions.eR00S02_NX3030_PlcA.abyBootloaderVersion[3]	:=	DG_NX4010.tRedundancy.RedUsrRem.abyUser[8]	;
		// Pocessador Auxiliar
		HwVersions.eR00S02_NX3030_PlcA.abyProcAuxVersion[0]	:=	DG_NX4010.tRedundancy.RedUsrRem.abyUser[9]	;
		HwVersions.eR00S02_NX3030_PlcA.abyProcAuxVersion[1]	:=	DG_NX4010.tRedundancy.RedUsrRem.abyUser[10]	;
		HwVersions.eR00S02_NX3030_PlcA.abyProcAuxVersion[2]	:=	DG_NX4010.tRedundancy.RedUsrRem.abyUser[11]	;
		HwVersions.eR00S02_NX3030_PlcA.abyProcAuxVersion[3]	:=	DG_NX4010.tRedundancy.RedUsrRem.abyUser[12]	;
		// Modelo CPU				
		HwVersions.eR00S02_NX3030_PlcA.dwCPUModel			:=	NonRedPointer.pdw02CPUModelRedUsrRem^	;
		// NX4010				
		HwVersions.eR00S04_NX4010_PlcA.dwFirmwareVersion	:=	NonRedPointer.pdw04NX4010FWRedUsrRem^	;
		HwVersions.eR00S04_NX4010_PlcA.dwProductID			:=	NonRedPointer.pdw04NX4010HWRedUsrRem^	;
		// NX50001				
		HwVersions.eR00S06_NX5001_PlcA.dwFirmwareVersion	:=	NonRedPointer.pdw06NX5001FWRedUsrRem^	;
		HwVersions.eR00S06_NX5001_PlcA.dwProductID			:=	NonRedPointer.pdw06NX5001HWRedUsrRem^	;
		HwVersions.eR00S08_NX5001_PlcA.dwFirmwareVersion	:=	NonRedPointer.pdw08NX5001FWRedUsrRem^	;
		HwVersions.eR00S08_NX5001_PlcA.dwProductID			:=	NonRedPointer.pdw08NX5001HWRedUsrRem^	;
		HwVersions.eR00S16_NX5001_PlcA.dwFirmwareVersion	:=	NonRedPointer.pdw16NX5001FWRedUsrRem^	;
		HwVersions.eR00S16_NX5001_PlcA.dwProductID			:=	NonRedPointer.pdw16NX5001HWRedUsrRem^	;
		// NX5000				
		HwVersions.eR00S10_NX5000_PlcA.dwFirmwareVersion	:=	NonRedPointer.pdw10NX5000FWRedUsrRem^	;
		HwVersions.eR00S10_NX5000_PlcA.dwProductID			:=	NonRedPointer.pdw10NX5000HWRedUsrRem^	;
		HwVersions.eR00S12_NX5000_PlcA.dwFirmwareVersion	:=	NonRedPointer.pdw12NX5000FWRedUsrRem^	;
		HwVersions.eR00S12_NX5000_PlcA.dwProductID			:=	NonRedPointer.pdw12NX5000HWRedUsrRem^	;
		HwVersions.eR00S20_NX5000_PlcA.dwFirmwareVersion	:=	NonRedPointer.pdw20NX5000FWRedUsrRem^	;
		HwVersions.eR00S20_NX5000_PlcA.dwProductID			:=	NonRedPointer.pdw20NX5000HWRedUsrRem^	;

	ELSIF	DG_NX4010.tRedundancy.RedDgnLoc.sGeneral_Diag.eRedState = REDUNDANCY_STATE.STANDBY	OR
			DG_NX4010.tRedundancy.RedDgnLoc.sGeneral_Diag.eRedState = REDUNDANCY_STATE.INACTIVE	THEN
		// Copia os dados deste PLC para a área de usuário do PLC remoto			
		// Firmware da CPU
		DG_NX4010.tRedundancy.RedUsrLoc.abyUser[1]	:=	HwVersions.eR00S02_NX3030_PlcB.abyCPUVersion[0]	;
		DG_NX4010.tRedundancy.RedUsrLoc.abyUser[2]	:=	HwVersions.eR00S02_NX3030_PlcB.abyCPUVersion[1]	;
		DG_NX4010.tRedundancy.RedUsrLoc.abyUser[3]	:=	HwVersions.eR00S02_NX3030_PlcB.abyCPUVersion[2]	;
		DG_NX4010.tRedundancy.RedUsrLoc.abyUser[4]	:=	HwVersions.eR00S02_NX3030_PlcB.abyCPUVersion[3]	;
		// Bootloader
		DG_NX4010.tRedundancy.RedUsrLoc.abyUser[5]	:=	HwVersions.eR00S02_NX3030_PlcB.abyBootloaderVersion[0]	;
		DG_NX4010.tRedundancy.RedUsrLoc.abyUser[6]	:=	HwVersions.eR00S02_NX3030_PlcB.abyBootloaderVersion[1]	;
		DG_NX4010.tRedundancy.RedUsrLoc.abyUser[7]	:=	HwVersions.eR00S02_NX3030_PlcB.abyBootloaderVersion[2]	;
		DG_NX4010.tRedundancy.RedUsrLoc.abyUser[8]	:=	HwVersions.eR00S02_NX3030_PlcB.abyBootloaderVersion[3]	;
		// Pocessador Auxiliar
		DG_NX4010.tRedundancy.RedUsrLoc.abyUser[9]	:=	HwVersions.eR00S02_NX3030_PlcB.abyProcAuxVersion[0]	;
		DG_NX4010.tRedundancy.RedUsrLoc.abyUser[10]	:=	HwVersions.eR00S02_NX3030_PlcB.abyProcAuxVersion[1]	;
		DG_NX4010.tRedundancy.RedUsrLoc.abyUser[11]	:=	HwVersions.eR00S02_NX3030_PlcB.abyProcAuxVersion[2]	;
		DG_NX4010.tRedundancy.RedUsrLoc.abyUser[12]	:=	HwVersions.eR00S02_NX3030_PlcB.abyProcAuxVersion[3]	;		
		// Modelo CPU
		NonRedPointer.pdw02CPUModelRedUsrLoc^	:=	HwVersions.eR00S02_NX3030_PlcB.dwCPUModel	;
		// NX4010
		NonRedPointer.pdw04NX4010FWRedUsrLoc^	:=	HwVersions.eR00S04_NX4010_PlcB.dwFirmwareVersion	;
		NonRedPointer.pdw04NX4010HWRedUsrLoc^	:=	HwVersions.eR00S04_NX4010_PlcB.dwProductID	;
		// NX50001
		NonRedPointer.pdw06NX5001FWRedUsrLoc^	:=	HwVersions.eR00S06_NX5001_PlcB.dwFirmwareVersion	;
		NonRedPointer.pdw06NX5001HWRedUsrLoc^	:=	HwVersions.eR00S06_NX5001_PlcB.dwProductID	;
		NonRedPointer.pdw08NX5001FWRedUsrLoc^	:=	HwVersions.eR00S08_NX5001_PlcB.dwFirmwareVersion	;
		NonRedPointer.pdw08NX5001HWRedUsrLoc^	:=	HwVersions.eR00S08_NX5001_PlcB.dwProductID	;
		NonRedPointer.pdw16NX5001FWRedUsrLoc^	:=	HwVersions.eR00S16_NX5001_PlcB.dwFirmwareVersion	;
		NonRedPointer.pdw16NX5001HWRedUsrLoc^	:=	HwVersions.eR00S16_NX5001_PlcB.dwProductID	;
		// NX5000
		NonRedPointer.pdw10NX5000FWRedUsrLoc^	:=	HwVersions.eR00S10_NX5000_PlcB.dwFirmwareVersion	;
		NonRedPointer.pdw10NX5000HWRedUsrLoc^	:=	HwVersions.eR00S10_NX5000_PlcB.dwProductID	;
		NonRedPointer.pdw12NX5000FWRedUsrLoc^	:=	HwVersions.eR00S12_NX5000_PlcB.dwFirmwareVersion	;
		NonRedPointer.pdw12NX5000HWRedUsrLoc^	:=	HwVersions.eR00S12_NX5000_PlcB.dwProductID	;
		NonRedPointer.pdw20NX5000FWRedUsrLoc^	:=	HwVersions.eR00S20_NX5000_PlcB.dwFirmwareVersion	;
		NonRedPointer.pdw20NX5000HWRedUsrLoc^	:=	HwVersions.eR00S20_NX5000_PlcB.dwProductID	;
		
	END_IF
END_IF

// Registra o tempo do sistema
SysTimeGetUs(uliPouEndTime);
// Calcula duração mínima/máxima desta POU
MinMaxTimes.uliPouMinTime_WriteHwVersionsNonActive:= MIN(MinMaxTimes.uliPouMinTime_WriteHwVersionsNonActive, uliPouEndTime - uliPouIniTime);
MinMaxTimes.uliPouMaxTime_WriteHwVersionsNonActive:= MAX(MinMaxTimes.uliPouMaxTime_WriteHwVersionsNonActive, uliPouEndTime - uliPouIniTime);

END_PROGRAM

// Device/Application/UserPOUs/Non-Redundant/MQTT
PROGRAM MQTT
VAR
// #######################################################################################	
	// Function Block -> Library LibMQTT	
	MQTT: LibMQTT.MQTT_CLIENT;
	CONN: LibMQTT.MQTT_CONN_CONFIG;
	SUBS: ARRAY [1..LibMQTT.gc_uiMaxSubs] OF LibMQTT.MQTT_SUBSCRIBE;
	PUBS: ARRAY [1..LibMQTT.gc_uiMaxPubs] OF LibMQTT.MQTT_PUBLISH;
	RCV: ARRAY [1..LibMQTT.gc_uiMaxSubs] OF LibMQTT.MQTT_RECEIVED;
	ENABLE: BOOL := TRUE; // Sempre vem habilitado o MQTT
	
	// Mensagem recebiba pelo subscriber
	sub1_RcvMessage : STRING;
	
	pub1_PubMessage : STRING;
	pub2_PubMessage : STRING;
	
	// Comando para disparar a publicação
	pub1_bEnablePublish : BOOL;
	pub2_bEnablePublish : BOOL;
	
	uliPouIniTime : ULINT;
	uliPouEndTime : ULINT;
END_VAR

// Registra o tempo do sistema
SysTimeGetUs(uliPouIniTime);

// Parâmetros de conexão com o Servidor A
CONN.bCleanSession :=TRUE;
CONN.sHostname := '192.168.16.86';
CONN.uiPort := 1883;       // Quando usado TLS porta deve ser 8883, caso contrário 1883.
CONN.uiKeepAlive := 60;
CONN.bEnableTLS := FALSE; // NX3010/20/30 não suportam TLS
CONN.sCertFilename := 'ca.crt';

// Parâmetros do Subscriber
SUBS[1].sSubscribeTopic := 'altus/jg03_NX3030/ElapsedTimeToFailure';
SUBS[1].eSubscribeQoS := LibMQTT.MQTT_QOS_2;
SUBS[1].pbPayloadBuffer := ADR(sub1_RcvMessage);
SUBS[1].uiMaxPayloadSize := SIZEOF(sub1_RcvMessage);

//Parâmetros do Publisher
PUBS[1].bEnablePublish := pub1_bEnablePublish AND NOT(MQTT.PUBLISH_STATUS[1]);
PUBS[1].sPublishTopic := 'altus/jg03_NX3030/ElapsedTimeToFailure';
PUBS[1].pbPublishPayload := ADR(pub1_PubMessage);
PUBS[1].uiPublishPayloadSize := INT_TO_UINT(LEN(pub1_PubMessage));
PUBS[1].ePublishMessageQoS := LibMQTT.MQTT_QOS_2;

//Parâmetros do Publisher
PUBS[2].bEnablePublish := pub2_bEnablePublish AND NOT(MQTT.PUBLISH_STATUS[2]);
PUBS[2].sPublishTopic := 'altus/jg03_NX3030/ElapsedTimeToFailureToScada';
PUBS[2].pbPublishPayload := ADR(pub2_PubMessage);
PUBS[2].uiPublishPayloadSize := INT_TO_UINT(LEN(pub2_PubMessage));
PUBS[2].ePublishMessageQoS := LibMQTT.MQTT_QOS_2;

// Chamada da função MQTT	
MQTT.ENABLE :=  (TRUE AND NOT(MQTT.ERROR));
MQTT.CONNECTION_CONFIG := CONN;
MQTT.SUBSCRIBE := SUBS;
MQTT.PUBLISH := PUBS;


// Somente chama a função se estiver no controlador correto.
// Essa consistência é devido ao pessoal do mtool utilizar projetos do superteste em outras CPUs.
IF (DG_NX3030.tDetailed.Ethernet.NET1.abyMAC[0] = 16#00 AND
	DG_NX3030.tDetailed.Ethernet.NET1.abyMAC[1] = 16#80 AND
	DG_NX3030.tDetailed.Ethernet.NET1.abyMAC[2] = 16#A0 AND
	DG_NX3030.tDetailed.Ethernet.NET1.abyMAC[3] = 16#05 AND
	DG_NX3030.tDetailed.Ethernet.NET1.abyMAC[4] = 16#F1 AND
	DG_NX3030.tDetailed.Ethernet.NET1.abyMAC[5] = 16#84) THEN
	MQTT();
END_IF


// Mensagem a ser publicada

// Para testar o MQTT por completo, uma mensagem é publicada no servidor,
// a mesma é lida pelo subscriber, e então enviado pelo segundo publisher que é mostrada na tela do SCADA
pub1_PubMessage := TIME_TO_STRING(PersistentVars.tElapsedTimeToFailure);
pub2_PubMessage:= sub1_RcvMessage;

// Dispara a publicação a cada 1 segundo, caso não tenha problemas de comunicação
IF MQTT.CONNECTED = TRUE AND 
	MQTT.STATE = LibMQTT.MQTT_STATES.MQTT_READY AND
	MQTT.ERROR = FALSE THEN
	
	pub1_bEnablePublish:= Special_Variables.Pulse_1s;
	pub2_bEnablePublish:= Special_Variables.Pulse_1s;
END_IF


// Registra o tempo do sistema
SysTimeGetUs(uliPouEndTime);
// Calcula duração mínima/máxima desta POU
MinMaxTimes.uliPouMinTime_MQTT:= MIN(MinMaxTimes.uliPouMinTime_MQTT, uliPouEndTime - uliPouIniTime);
MinMaxTimes.uliPouMaxTime_MQTT:= MAX(MinMaxTimes.uliPouMaxTime_MQTT, uliPouEndTime - uliPouIniTime);

END_PROGRAM

// Device/Application/UserPOUs/Non-Redundant/CleanStats
PROGRAM CleanStats
VAR
	uliPouIniTime : ULINT;
	uliPouEndTime : ULINT;
END_VAR
VAR RETAIN
	iCleanStatsCallCnt : INT := 0;
END_VAR

// POU que zera o relatório dos testes, que é retentivo.
// Precisa ser habilitada na ActivePrg.

// Registra o tempo do sistema
SysTimeGetUs(uliPouIniTime);

// Registra a chamada desta POU
iCleanStatsCallCnt:= iCleanStatsCallCnt + 1;

// Solicita reinicialização dos contadores do MODBUS
DG_MODBUS_Master_1.tCommand.bResetCounter:= TRUE;
DG_MODBUS_Slave_1.tCommand.bResetCounter:= TRUE;
DG_MODBUS_Client_2.tCommand.bResetCounter:= TRUE;
DG_MODBUS_Server_2.tCommand.bResetCounter:= TRUE;
DG_MODBUS_Client_3.tCommand.bResetCounter:= TRUE;
DG_MODBUS_Server_3.tCommand.bResetCounter:= TRUE;
DG_MODBUS_Client_4.tCommand.bResetCounter:= TRUE;
DG_MODBUS_Server_4.tCommand.bResetCounter:= TRUE;
// Solicita reinicialização dos contadores do NX4010
DG_NX4010.tRedundancy.RedCmdLoc.bResetNETStatisticsLocal:= TRUE;
DG_NX4010.tRedundancy.RedCmdLoc.bResetNETStatisticsRemote:= TRUE;
// Resultados da POU StateChange:
Persistentvars.bExchangeStateFail:= FALSE;
Persistentvars.dwTransitionsCnt:= 0;
Persistentvars.dwSwitchoverCnt:= 0;
// Resultados das POUs CheckRedData e IncrRedData:
Persistentvars.iSyncFailCntSymb:= 0;
Persistentvars.iSyncFailCntQ:= 0;
Persistentvars.iSyncFailCntM:= 0;
Persistentvars.iSyncFailCntI:= 0;
PersistentVars.iSyncFailCallback_vfInit :=0;
NonRedPointer.piSSyncFailLoc^:= 0;
NonRedPointer.piQSyncFailLoc^:= 0;
NonRedPointer.piMSyncFailLoc^:= 0;
NonRedPointer.piISyncFailLoc^:= 0;
NonRedPointer.piSSyncFailRem^:= 0;
NonRedPointer.piQSyncFailRem^:= 0;
NonRedPointer.piMSyncFailRem^:= 0;
NonRedPointer.piISyncFailRem^:= 0;
// Resultados da POU CycleTimes:
Symbolics.bPlcAMaxMinSetup:= TRUE;
Persistentvars.dwPLCAMainTaskLoadMax:= 0;	
Persistentvars.dwPLCAMainTaskLoadAvg:= 0;	
Persistentvars.dwPLCAMainTaskLoadMin:= 10000; 	
Symbolics.bPlcBMaxMinSetup:= TRUE;
Persistentvars.dwPLCBMainTaskLoadMax:= 0;
Persistentvars.dwPLCBMainTaskLoadAvg:= 0;	
Persistentvars.dwPLCBMainTaskLoadMin:= 10000;
// Resultados da POU CheckProfibusIOs:
Persistentvars.dwSlave5DigIOsErrors:= 0;
Persistentvars.dwSlave5Unavailable:= 0;
Persistentvars.dwSlave5ModulesOut:= 0;
Persistentvars.dwSlave10AnaIOsErrors:= 0;
Persistentvars.dwSlave10Unavailable:= 0;
Persistentvars.dwSlave10ModulesOut:= 0;
Persistentvars.dwSlave3DigIOsErrors:= 0;
Persistentvars.dwSlave3Unavailable:= 0;
Persistentvars.dwSlave3ModulesOut:= 0;
PersistentVars.wErrorValuePO2132C00:= 0;
PersistentVars.wErrorValuePO1212C00:= 0;
PersistentVars.bFrozenErrorRem05TORem05:= FALSE;
PersistentVars.bFrozenErrorRem05TORem04:= FALSE;
// CheckModbus1
Persistentvars.bModbus1ErrorCoil:= FALSE;
Persistentvars.bModbus1ErrorStatus:= FALSE;
Persistentvars.bModbus1ErrorHolding:= FALSE;
Persistentvars.bModbus1ErrorInputReg:= FALSE;
NonRedPointer.pbModbus1ErrorCoilLoc^:= FALSE;
NonRedPointer.pbModbus1ErrorCoilRem^:= FALSE;
NonRedPointer.pbModbus1ErrorStatusLoc^:= FALSE;
NonRedPointer.pbModbus1ErrorStatusRem^:= FALSE;
NonRedPointer.pbModbus1ErrorHoldingLoc^:= FALSE;
NonRedPointer.pbModbus1ErrorHoldingRem^:= FALSE;
NonRedPointer.pbModbus1ErrorInputRegLoc^:= FALSE;
NonRedPointer.pbModbus1ErrorInputRegRem^:= FALSE;
// CheckModbus2
Persistentvars.bModbus2ErrorCoil:= FALSE;
Persistentvars.bModbus2ErrorStatus:= FALSE;
Persistentvars.bModbus2ErrorHolding:= FALSE;
Persistentvars.bModbus2ErrorInputReg:= FALSE;
// CheckModbus3
Persistentvars.bModbus3ErrorCoil:= FALSE;
Persistentvars.bModbus3ErrorStatus:= FALSE;
Persistentvars.bModbus3ErrorHolding:= FALSE;
Persistentvars.bModbus3ErrorInputReg:= FALSE;
// CheckModbus4
Persistentvars.bModbus4ErrorCoil:= FALSE;
Persistentvars.bModbus4ErrorStatus:= FALSE;
Persistentvars.bModbus4ErrorHolding:= FALSE;
Persistentvars.bModbus4ErrorInputReg:= FALSE;

// Resultados da POU SOE:
Persistentvars.bSOE1EventsMismatch:= FALSE;
Persistentvars.bSOE1FalseOverflow:= FALSE;
Persistentvars.bSOE2EventsMismatch:= FALSE;
Persistentvars.bSOE2FalseOverflow:= FALSE;

// Resultados POU UserLog
NonRedData.iStepUserlog:=0;	
NonRedPointer.pbErrorUserLogLoc^ := FALSE;
NonRedPointer.pbErrorUserLogRem^ := FALSE;
PersistentVars.bUserLog := FALSE;
//Resultados POU Languages
PersistentVars.dwErrorLanguages:= 0;


// Resultados POU ProfibusStateChange
PersistentVars.dwPBSwitchoverCnt:= 0;

// Resultados da POU SNTP_PLCx:
PersistentVars.bSntpServerFailures:= FALSE;
PersistentVars.bSntpSourceFailures:= FALSE;
PersistentVars.bTimezoneFailure := FALSE;
PersistentVars.iSntpSyncFailures:= 0;

// Resultados da POU CheckRam
PersistentVars.bRamTotalFailure:= FALSE;
PersistentVars.bRamFreeVarFailure:= FALSE;
PersistentVars.dwMinFreeRamPlcA:= 95832; //Atualizado em 12/08/2019
PersistentVars.dwMaxFreeRamPlcA:= 0;
PersistentVars.dwMinFreeRamPlcB:= 95832; //Atualizado em 12/08/2019
PersistentVars.dwMaxFreeRamPlcB:= 0;

// Tempos mínimos/médio/máximo da NonSkippedPrg e ActivePrg (UCP redundante)
MinMaxTimes.uliPouMinTime_NonSkippedPrg:=			65535;
MinMaxTimes.uliPouMaxTime_NonSkippedPrg:=			0;
MinMaxTimes.uliPouMinTime_ActivePrg:=				65535;
MinMaxTimes.uliPouMaxTime_ActivePrg:=				0;

// Tempos mínimos/máximos de duração das POUs
MinMaxTimes.uliPouMinTime_Alarms:=					65535;
MinMaxTimes.uliPouMaxTime_Alarms:= 					0;
MinMaxTimes.uliPouMinTime_CheckDiags:=				65535;
MinMaxTimes.uliPouMaxTime_CheckDiags:=				0;
MinMaxTimes.uliPouMinTime_CheckIec104:=				65535;
MinMaxTimes.uliPouMaxTime_CheckIec104:=				0;
MinMaxTimes.uliPouMinTime_CheckLanguages:=			65535;
MinMaxTimes.uliPouMaxTime_CheckLanguages:=			0;
MinMaxTimes.uliPouMinTime_CheckModbus1:=			65535;
MinMaxTimes.uliPouMaxTime_CheckModbus1:=			0;
MinMaxTimes.uliPouMinTime_CheckModbus2:=			65535;
MinMaxTimes.uliPouMaxTime_CheckModbus2:=			0;
MinMaxTimes.uliPouMinTime_CheckModbus3:=			65535;
MinMaxTimes.uliPouMaxTime_CheckModbus3:=			0;
MinMaxTimes.uliPouMinTime_CheckModbus4:=			65535;
MinMaxTimes.uliPouMaxTime_CheckModbus4:=			0;
MinMaxTimes.uliPouMinTime_CheckProfibusIOs:=		65535;
MinMaxTimes.uliPouMaxTime_CheckProfibusIOs:=		0;
MinMaxTimes.uliPouMinTime_CheckRecipe:=				65535;
MinMaxTimes.uliPouMaxTime_CheckRecipe:=				0;
MinMaxTimes.uliPouMinTime_CheckRedData:=			65535;
MinMaxTimes.uliPouMaxTime_CheckRedData:=			0;
MinMaxTimes.uliPouMinTime_CheckSntp:=				65535;
MinMaxTimes.uliPouMaxTime_CheckSntp:=				0;
MinMaxTimes.uliPouMinTime_CheckSoe:=				65535;
MinMaxTimes.uliPouMaxTime_CheckSoe:=				0;
MinMaxTimes.uliPouMinTime_CheckSpecialVars:=		65535;
MinMaxTimes.uliPouMaxTime_CheckSpecialVars:=		0;
MinMaxTimes.uliPouMinTime_CleanStatus:=				MinMaxTimes.uliPouMinTime_CleanStatus;	// Não inicializar com 65535
MinMaxTimes.uliPouMaxTime_CleanStatus:=				MinMaxTimes.uliPouMaxTime_CleanStatus;	// Não inicializar com 0
MinMaxTimes.uliPouMinTime_CycleTimes:=				65535;
MinMaxTimes.uliPouMaxTime_CycleTimes:=				0;
MinMaxTimes.uliPouMinTime_IncrRedData:=				65535;
MinMaxTimes.uliPouMaxTime_IncrRedData:=				0;
MinMaxTimes.uliPouMinTime_DaylightSavingTime:=		65535;
MinMaxTimes.uliPouMaxTime_DaylightSavingTime:=		0;
MinMaxTimes.uliPouMinTime_PidGenerator:=			65535;
MinMaxTimes.uliPouMaxTime_PidGenerator:=			0;
MinMaxTimes.uliPouMinTime_StateChange:=				65535;
MinMaxTimes.uliPouMaxTime_StateChange:=				0;
MinMaxTimes.uliPouMinTime_UserLog:=					65535;
MinMaxTimes.uliPouMaxTime_UserLog:=					0;
MinMaxTimes.uliPouMinTime_CheckRam:=				65535;
MinMaxTimes.uliPouMaxTime_CheckRam:=				0;
MinMaxTimes.uliPouMinTime_CheckForcing:= 			65535;
MinMaxTimes.uliPouMaxTime_CheckForcing:=			 0;
MinMaxTimes.uliPouMinTime_WriteHwVersionsNonActive:=65535;
MinMaxTimes.uliPouMaxTime_WriteHwVersionsNonActive:=0;
MinMaxTimes.uliPouMinTime_CheckNVL:=				65535;
MinMaxTimes.uliPouMaxTime_CheckNVL:=				0;
MinMaxTimes.uliPouMinTime_MQTT:=					65535;
MinMaxTimes.uliPouMaxTime_MQTT:=					0;


// Tempos MÁXIMOS de transição das entradas que são imagem/cópia das saídas
MinMaxTimes.liDigMaxTime_CheckModbus1:=				0;
MinMaxTimes.liAnaMaxTime_CheckModbus1:=				0;
MinMaxTimes.liDigMaxTime_CheckModbus2:=				0;
MinMaxTimes.liAnaMaxTime_CheckModbus2:=				0;
MinMaxTimes.liDigMaxTime_CheckModbus3:=				0;
MinMaxTimes.liAnaMaxTime_CheckModbus3:=				0;
MinMaxTimes.liDigMaxTime_CheckModbus4:=				0;
MinMaxTimes.liAnaMaxTime_CheckModbus4:=				0;
MinMaxTimes.liDigMaxTime_CheckProfibusIOs:=			0;
MinMaxTimes.liAnaMaxTime_CheckProfibusIOs:=			0;
MinMaxTimes.liNXMaxTime_CheckProfibusIOs:=			0;
MinMaxTimes.liAna99MaxTime_CheckProfibusIOs:=		0;
MinMaxTimes.liDig99MaxTime_CheckProfibusIOs:=		0;
MinMaxTimes.liDig99MaxTime1005_CheckProfibusIOs:=	0;

// Limpa Diagnósticos utilizados na CheckDiags
	// NX3030
	DiagsRetain.DG_NX3030_tSummarized_bAbsentModules:= 0;
	DiagsRetain.DG_NX3030_tSummarized_bAbsentRacks:= 0;
	DiagsRetain.DG_NX3030_tSummarized_bCOM1ConfigError:= 0;
	DiagsRetain.DG_NX3030_tSummarized_bCOM2ConfigError:= 0;
	DiagsRetain.DG_NX3030_tSummarized_bConfigMismatch:= 0;
	DiagsRetain.DG_NX3030_tSummarized_bDuplicatedRacks:= 0;
	DiagsRetain.DG_NX3030_tSummarized_bDuplicatedSlots:= 0;
	DiagsRetain.DG_NX3030_tSummarized_bHardwareFailure:= 0;
	DiagsRetain.DG_NX3030_tSummarized_bInvalidDateTime:= 0;
	DiagsRetain.DG_NX3030_tSummarized_bInvalidRacks:= 0;
	DiagsRetain.DG_NX3030_tSummarized_bMemoryCardError:= 0;
	DiagsRetain.DG_NX3030_tSummarized_bModuleFatalError:= 0;
	DiagsRetain.DG_NX3030_tSummarized_bModuleParameterError:= 0;
	DiagsRetain.DG_NX3030_tSummarized_bModulesWithDiagnostic:= 0;
	DiagsRetain.DG_NX3030_tSummarized_bNET1ConfigError:= 0;
	DiagsRetain.DG_NX3030_tSummarized_bNET2ConfigError:= 0;
	DiagsRetain.DG_NX3030_tSummarized_bNonDeclaredModules:= 0;
	DiagsRetain.DG_NX3030_tSummarized_bNonDeclaredRacks:= 0;
	DiagsRetain.DG_NX3030_tSummarized_bOTDSwitchError:= 0;
	DiagsRetain.DG_NX3030_tSummarized_bRuntimeReset:= 0;
	DiagsRetain.DG_NX3030_tSummarized_bSoftwareException:= 0;
	DiagsRetain.DG_NX3030_tSummarized_bSwappedModules:= 0;
	DiagsRetain.DG_NX3030_tSummarized_bWHSBBusError:= 0;
	DiagsRetain.DG_NX3030_tDetailed_MemoryCard_byMounted:= 0;
	DiagsRetain.DG_NX3030_tDetailed_Ethernet_NET1_bLinkDown:= 0;
	DiagsRetain.DG_NX3030_tDetailed_Ethernet_NET2_bLinkDown:= 0;	
	DiagsRetain.DG_NX3030_tDetailed_Application_byCPUState := 0;
	DiagsRetain.DG_NX3030_tDetailed_ApplicationInfo_dwApplicationCRC := 0;
	DiagsRetain.DG_NX3030_tDetailed_Ethernet_NET1_abyMAC_0 := 0;
	DiagsRetain.DG_NX3030_tDetailed_Ethernet_NET1_abyMAC_1 := 0;
	DiagsRetain.DG_NX3030_tDetailed_Ethernet_NET1_abyMAC_2 := 0;
	DiagsRetain.DG_NX3030_tDetailed_Ethernet_NET1_abyMAC_3 := 0;
	DiagsRetain.DG_NX3030_tDetailed_Ethernet_NET1_abyMAC_4 := 0;
	DiagsRetain.DG_NX3030_tDetailed_Ethernet_NET1_abyMAC_5 := 0;
	DiagsRetain.DG_NX3030_tDetailed_Ethernet_NET2_abyMAC_0 := 0;
	DiagsRetain.DG_NX3030_tDetailed_Ethernet_NET2_abyMAC_1 := 0;
	DiagsRetain.DG_NX3030_tDetailed_Ethernet_NET2_abyMAC_2 := 0;
	DiagsRetain.DG_NX3030_tDetailed_Ethernet_NET2_abyMAC_3 := 0;
	DiagsRetain.DG_NX3030_tDetailed_Ethernet_NET2_abyMAC_4 := 0;
	DiagsRetain.DG_NX3030_tDetailed_Ethernet_NET2_abyMAC_5 := 0;
	DiagsRetain.DG_NX3030_tDetailed_Ethernet_NETx_abyIP_0 := 0;
	DiagsRetain.DG_NX3030_tDetailed_Ethernet_NETx_abyIP_1 := 0;
	DiagsRetain.DG_NX3030_tDetailed_Ethernet_NETx_abyIP_2 := 0;
	DiagsRetain.DG_NX3030_tDetailed_Ethernet_NETx_abyIP_3 := 0;
	DiagsRetain.DG_NX3030_tDetailed_Ethernet_NETx_abyMask_0 := 0;
	DiagsRetain.DG_NX3030_tDetailed_Ethernet_NETx_abyMask_1 := 0;
	DiagsRetain.DG_NX3030_tDetailed_Ethernet_NETx_abyMask_2 := 0;
	DiagsRetain.DG_NX3030_tDetailed_Ethernet_NETx_abyMask_3 := 0;
	DiagsRetain.DG_NX3030_tDetailed_Ethernet_NETx_abyGateway_0 := 0;
	DiagsRetain.DG_NX3030_tDetailed_Ethernet_NETx_abyGateway_1 := 0;
	DiagsRetain.DG_NX3030_tDetailed_Ethernet_NETx_abyGateway_2 := 0;
	DiagsRetain.DG_NX3030_tDetailed_Ethernet_NETx_abyGateway_3 := 0;
	DiagsRetain.DG_NX3030_tDetailed_SNTP_bServiceEnabled := 0;
	DiagsRetain.DG_NX3030_tDetailed_Target_abyAuxprocVersion := 0;
	DiagsRetain.DG_NX3030_tDetailed_Target_abyBootloaderVersion := 0;
	DiagsRetain.DG_NX3030_tDetailed_Target_abyCPUVersion := 0;
	DiagsRetain.DG_NX3030_tDetailed_Target_dwCPUModel := 0;
	DiagsRetain.DG_NX3030_tDetailed_Thermometer_diTemperature := 0;
	// NX4010
	DiagsRetain.DG_NX4010_tGeneral_bActiveDiagnostics:= 0;
	DiagsRetain.DG_NX4010_tGeneral_bBusCommunicationError:= 0;
	DiagsRetain.DG_NX4010_tGeneral_bConfigMismatch:= 0;
	DiagsRetain.DG_NX4010_tGeneral_bFatalError:= 0;
	DiagsRetain.DG_NX4010_tGeneral_bNET1LinkDown:= 0;
	DiagsRetain.DG_NX4010_tGeneral_bNET2LinkDown:= 0;
	DiagsRetain.DG_NX4010_tGeneral_bOTDSwitchError:= 0;
	DiagsRetain.DG_NX4010_tGeneral_bWatchdogError:= 0;
	DiagsRetain.DG_NX4010_tRedundancy_RedDgnLoc_sGeneral_Diag_bApplicationIncompatible:= 0;
	DiagsRetain.DG_NX4010_tRedundancy_RedDgnLoc_sGeneral_Diag_bApplicationProjectDiff:= 0;
	DiagsRetain.DG_NX4010_tRedundancy_RedDgnLoc_sGeneral_Diag_bConfigError:= 0;
	DiagsRetain.DG_NX4010_tRedundancy_RedDgnLoc_sGeneral_Diag_bExchangeSync:= 0;
	DiagsRetain.DG_NX4010_tRedundancy_RedDgnLoc_sGeneral_Diag_bFailedPBUS1A:= 0;
	DiagsRetain.DG_NX4010_tRedundancy_RedDgnLoc_sGeneral_Diag_bFailedPBUS1B:= 0;
	DiagsRetain.DG_NX4010_tRedundancy_RedDgnLoc_sGeneral_Diag_bFailedPBUS2A:= 0;
	DiagsRetain.DG_NX4010_tRedundancy_RedDgnLoc_sGeneral_Diag_bFailedPBUS2B:= 0;
	DiagsRetain.DG_NX4010_tRedundancy_RedDgnLoc_sGeneral_Diag_bFailedRED:= 0;
	DiagsRetain.DG_NX4010_tRedundancy_RedDgnLoc_sGeneral_Diag_bFailureProfibus_1:= 0;
	DiagsRetain.DG_NX4010_tRedundancy_RedDgnLoc_sGeneral_Diag_bFailureProfibus_2:= 0;
	DiagsRetain.DG_NX4010_tRedundancy_RedDgnLoc_sGeneral_Diag_bIncompatibleFirmware:= 0;
	DiagsRetain.DG_NX4010_tRedundancy_RedDgnLoc_sGeneral_Diag_bProfibusVitalFailureAll:= 0;
	DiagsRetain.DG_NX4010_tRedundancy_RedDgnLoc_sGeneral_Diag_bProfibusVitalFailureAny:= 0;
	DiagsRetain.DG_NX4010_tRedundancy_RedDgnLoc_sGeneral_Diag_bProjectArchiveDiff:= 0;
	DiagsRetain.DG_NX4010_tRedundancy_RedDgnLoc_sGeneral_Diag_bProjectSyncDisable:= 0;
	DiagsRetain.DG_NX4010_tRedundancy_RedDgnLoc_sGeneral_Diag_bRedDataSync:= 0;
	DiagsRetain.DG_NX4010_tRedundancy_RedDgnLoc_sGeneral_Diag_bRedForceSync:= 0;
	DiagsRetain.DG_NX4010_tRedundancy_RedDgnLoc_sGeneral_Diag_bRedPanelTestMode:= 0;
	DiagsRetain.DG_NX4010_tRedundancy_RedDgnLoc_sGeneral_Diag_bTemporaryBufferTooSmall:= 0;
	DiagsRetain.DG_NX4010_tRedundancy_RedDgnLoc_sGeneral_Diag_bTooManyRedAreas:= 0;
	DiagsRetain.DG_NX4010_tRedundancy_RedDgnLoc_sGeneral_Diag_dwApplicationCRC:= 0;
	DiagsRetain.DG_NX4010_tRedundancy_RedDgnLoc_sGeneral_Diag_dwArchiveCRC:= 0;
	// NX5001_1
	DiagsRetain.DG_NX5001_1_tGeneral_bActiveDiagnostics:= 0;
	DiagsRetain.DG_NX5001_1_tGeneral_bBusCommunicationError:= 0;
	DiagsRetain.DG_NX5001_1_tGeneral_bConfigMismatch:= 0;
	DiagsRetain.DG_NX5001_1_tGeneral_bFatalError:= 0;
	DiagsRetain.DG_NX5001_1_tGeneral_bNX5001NoCfg:= 0;
	DiagsRetain.DG_NX5001_1_tGeneral_bOTDSwitchError:= 0;
	DiagsRetain.DG_NX5001_1_tGeneral_bPbusCommFail:= 0;
	DiagsRetain.DG_NX5001_1_tGeneral_bSlaveNotConfigured:= 0;
	DiagsRetain.DG_NX5001_1_tGeneral_bSlaveNotPresent:= 0;
	DiagsRetain.DG_NX5001_1_tGeneral_bSlaveWithDiagnostic:= 0;
	DiagsRetain.DG_NX5001_1_tGeneral_bStsEnableInterface:= 0;
	DiagsRetain.DG_NX5001_1_tGeneral_bStsMstRedundEnable:= 0;
	DiagsRetain.DG_NX5001_1_tGeneral_bWatchdogError:= 0;
	DiagsRetain.DG_NX5001_1_tMstStatus_abySlv_Diag_bSlave_5:= 0;
	DiagsRetain.DG_NX5001_1_tMstStatus_abySlv_Diag_bSlave_10:= 0;
	DiagsRetain.DG_NX5001_1_tMstStatus_abySlv_Diag_bSlave_99:= 0;

	// NX5001_2
	DiagsRetain.DG_NX5001_2_tGeneral_bActiveDiagnostics:= 0;
	DiagsRetain.DG_NX5001_2_tGeneral_bBusCommunicationError:= 0;
	DiagsRetain.DG_NX5001_2_tGeneral_bConfigMismatch:= 0;
	DiagsRetain.DG_NX5001_2_tGeneral_bFatalError:= 0;
	DiagsRetain.DG_NX5001_2_tGeneral_bNX5001NoCfg:= 0;
	DiagsRetain.DG_NX5001_2_tGeneral_bOTDSwitchError:= 0;
	DiagsRetain.DG_NX5001_2_tGeneral_bPbusCommFail:= 0;
	DiagsRetain.DG_NX5001_2_tGeneral_bSlaveNotConfigured:= 0;
	DiagsRetain.DG_NX5001_2_tGeneral_bSlaveNotPresent:= 0;
	DiagsRetain.DG_NX5001_2_tGeneral_bSlaveWithDiagnostic:= 0;
	DiagsRetain.DG_NX5001_2_tGeneral_bStsEnableInterface:= 0;
	DiagsRetain.DG_NX5001_2_tGeneral_bStsMstRedundEnable:= 0;
	DiagsRetain.DG_NX5001_2_tGeneral_bWatchdogError:= 0;
	DiagsRetain.DG_NX5001_2_tMstStatus_abySlv_Diag_bSlave_5:= 0;
	DiagsRetain.DG_NX5001_2_tMstStatus_abySlv_Diag_bSlave_10:= 0;
	DiagsRetain.DG_NX5001_2_tMstStatus_abySlv_Diag_bSlave_99:= 0;
	// NX5001_3
	DiagsRetain.DG_NX5001_3_tGeneral_bActiveDiagnostics:= 0;
	DiagsRetain.DG_NX5001_3_tGeneral_bBusCommunicationError:= 0;
	DiagsRetain.DG_NX5001_3_tGeneral_bConfigMismatch:= 0;
	DiagsRetain.DG_NX5001_3_tGeneral_bFatalError:= 0;
	DiagsRetain.DG_NX5001_3_tGeneral_bNX5001NoCfg:= 0;
	DiagsRetain.DG_NX5001_3_tGeneral_bOTDSwitchError:= 0;
	DiagsRetain.DG_NX5001_3_tGeneral_bPbusCommFail:= 0;
	DiagsRetain.DG_NX5001_3_tGeneral_bSlaveNotConfigured:= 0;
	DiagsRetain.DG_NX5001_3_tGeneral_bSlaveNotPresent:= 0;
	DiagsRetain.DG_NX5001_3_tGeneral_bSlaveWithDiagnostic:= 0;
	DiagsRetain.DG_NX5001_3_tGeneral_bStsEnableInterface:= 0;
	DiagsRetain.DG_NX5001_3_tGeneral_bStsMstRedundEnable:= 0;
	DiagsRetain.DG_NX5001_3_tGeneral_bWatchdogError:= 0;
	DiagsRetain.DG_NX5001_3_tMstStatus_abySlv_Diag_bSlave_4:= 0;
	DiagsRetain.DG_NX5001_3_tMstStatus_abySlv_Diag_bSlave_99:= 0;
	// NX5000_1	
 	DiagsRetain.DG_NX5000_1_tGeneral_bActiveDiagnostics:= 0;
	DiagsRetain.DG_NX5000_1_tGeneral_bBusCommunicationError:= 0;
	DiagsRetain.DG_NX5000_1_tGeneral_bConfigMismatch:= 0;
	DiagsRetain.DG_NX5000_1_tGeneral_bFatalError:= 0;
	DiagsRetain.DG_NX5000_1_tGeneral_bOTDSwitchError:= 0;
	DiagsRetain.DG_NX5000_1_tGeneral_bWatchdogError:= 0;
	DiagsRetain.DG_NX5000_1_tNX5000_bNX5000NoCfg:= 0;
	DiagsRetain.DG_NX5000_1_tNX5000_bStsEthLink:= 0;
	// NX5000_2	
 	DiagsRetain.DG_NX5000_2_tGeneral_bActiveDiagnostics:= 0;
	DiagsRetain.DG_NX5000_2_tGeneral_bBusCommunicationError:= 0;
	DiagsRetain.DG_NX5000_2_tGeneral_bConfigMismatch:= 0;
	DiagsRetain.DG_NX5000_2_tGeneral_bFatalError:= 0;
	DiagsRetain.DG_NX5000_2_tGeneral_bOTDSwitchError:= 0;
	DiagsRetain.DG_NX5000_2_tGeneral_bWatchdogError:= 0;
	DiagsRetain.DG_NX5000_2_tNX5000_bNX5000NoCfg:= 0;
	DiagsRetain.DG_NX5000_2_tNX5000_bStsEthLink:= 0;
	// NX5000_3	
 	DiagsRetain.DG_NX5000_3_tGeneral_bActiveDiagnostics:= 0;
	DiagsRetain.DG_NX5000_3_tGeneral_bBusCommunicationError:= 0;
	DiagsRetain.DG_NX5000_3_tGeneral_bConfigMismatch:= 0;
	DiagsRetain.DG_NX5000_3_tGeneral_bFatalError:= 0;
	DiagsRetain.DG_NX5000_3_tGeneral_bOTDSwitchError:= 0;
	DiagsRetain.DG_NX5000_3_tGeneral_bWatchdogError:= 0;
	DiagsRetain.DG_NX5000_3_tNX5000_bNX5000NoCfg:= 0;
	DiagsRetain.DG_NX5000_3_tNX5000_bStsEthLink:= 0;
	// DiagsRetain.DG_MODBUS_Master_1
	DiagsRetain.DG_MODBUS_Master_1_tDiag_bConfigFailure:= 0;
	DiagsRetain.DG_MODBUS_Master_1_tDiag_bModuleFailure:= 0;
	DiagsRetain.DG_MODBUS_Master_1_tDiag_bRXFailure:= 0;
	DiagsRetain.DG_MODBUS_Master_1_tDiag_bTXFailure:= 0;
	// MODBUS_Slave_1	
	DiagsRetain.DG_MODBUS_Slave_1_tDiag_bConfigFailure:= 0;
	DiagsRetain.DG_MODBUS_Slave_1_tDiag_bModuleFailure:= 0;
	DiagsRetain.DG_MODBUS_Slave_1_tDiag_bRXFailure:= 0;
	DiagsRetain.DG_MODBUS_Slave_1_tDiag_bTXFailure:= 0;
	// MODBUS_Client_2
	DiagsRetain.DG_MODBUS_Client_2_tDiag_bConfigFailure:= 0;
	DiagsRetain.DG_MODBUS_Client_2_tDiag_bModuleFailure:= 0;
	DiagsRetain.DG_MODBUS_Client_2_tDiag_bRXFailure:= 0;
	DiagsRetain.DG_MODBUS_Client_2_tDiag_bTXFailure:= 0;
	// MODBUS_Server_2
	DiagsRetain.DG_MODBUS_Server_2_tDiag_bConfigFailure:= 0;
	DiagsRetain.DG_MODBUS_Server_2_tDiag_bModuleFailure:= 0;
	DiagsRetain.DG_MODBUS_Server_2_tDiag_bRXFailure:= 0;
	DiagsRetain.DG_MODBUS_Server_2_tDiag_bTXFailure:= 0;
	// MODBUS_Client_3
	DiagsRetain.DG_MODBUS_Client_3_tDiag_bConfigFailure:= 0;
	DiagsRetain.DG_MODBUS_Client_3_tDiag_bModuleFailure:= 0;
	DiagsRetain.DG_MODBUS_Client_3_tDiag_bRXFailure:= 0;
	DiagsRetain.DG_MODBUS_Client_3_tDiag_bTXFailure:= 0;
	// MODBUS_Server_3
	DiagsRetain.DG_MODBUS_Server_3_tDiag_bConfigFailure:= 0;
	DiagsRetain.DG_MODBUS_Server_3_tDiag_bModuleFailure:= 0;
	DiagsRetain.DG_MODBUS_Server_3_tDiag_bRXFailure:= 0;
	DiagsRetain.DG_MODBUS_Server_3_tDiag_bTXFailure:= 0;
	// MODBUS_Client_4
	DiagsRetain.DG_MODBUS_Client_4_tDiag_bConfigFailure:= 0;
	DiagsRetain.DG_MODBUS_Client_4_tDiag_bModuleFailure:= 0;
	DiagsRetain.DG_MODBUS_Client_4_tDiag_bRXFailure:= 0;
	DiagsRetain.DG_MODBUS_Client_4_tDiag_bTXFailure:= 0;
	// MODBUS_Server_4	
	DiagsRetain.DG_MODBUS_Server_4_tDiag_bConfigFailure:= 0;
	DiagsRetain.DG_MODBUS_Server_4_tDiag_bModuleFailure:= 0;
	DiagsRetain.DG_MODBUS_Server_4_tDiag_bRXFailure:= 0;
	DiagsRetain.DG_MODBUS_Server_4_tDiag_bTXFailure:= 0;
	
	//PO1000		
DiagsRetain.DG_REM05_PO1000_bHardwareFailure	:=	0;
DiagsRetain.DG_REM05_PO1000_bPowerSupplyFail	:=	0;
		
//PO2020		
DiagsRetain.DG_REM05_PO2020_bHardwareFailure	:=	0;
DiagsRetain.DG_REM05_PO2020_bPowerSupplyFail	:=	0;
		
//PO9100		
DiagsRetain.DG_REM05_PO9100_bReserved00	:=	0;
		
//PO1212		
DiagsRetain.DG_REM10_PO1212_bFuseOpen	:=	0;
DiagsRetain.DG_REM10_PO1212_bHardwareFailure	:=	0;
DiagsRetain.DG_REM10_PO1212_bNoParametrizedModule	:=	0;
DiagsRetain.DG_REM10_PO1212_bOverTemp	:=	0;
DiagsRetain.DG_REM10_PO1212_aCh0_bOpenSensor	:=	0;
DiagsRetain.DG_REM10_PO1212_aCh0_bOverRange	:=	0;
DiagsRetain.DG_REM10_PO1212_aCh0_bSensorShortCircuit	:=	0;
DiagsRetain.DG_REM10_PO1212_aCh0_bWrongParameters	:=	0;
DiagsRetain.DG_REM10_PO1212_aCh1_bOpenSensor	:=	0;
DiagsRetain.DG_REM10_PO1212_aCh1_bOverRange	:=	0;
DiagsRetain.DG_REM10_PO1212_aCh1_bSensorShortCircuit	:=	0;
DiagsRetain.DG_REM10_PO1212_aCh1_bWrongParameters	:=	0;
DiagsRetain.DG_REM10_PO1212_aCh2_bOpenSensor	:=	0;
DiagsRetain.DG_REM10_PO1212_aCh2_bOverRange	:=	0;
DiagsRetain.DG_REM10_PO1212_aCh2_bSensorShortCircuit	:=	0;
DiagsRetain.DG_REM10_PO1212_aCh2_bWrongParameters	:=	0;
DiagsRetain.DG_REM10_PO1212_aCh3_bOpenSensor	:=	0;
DiagsRetain.DG_REM10_PO1212_aCh3_bOverRange	:=	0;
DiagsRetain.DG_REM10_PO1212_aCh3_bSensorShortCircuit	:=	0;
DiagsRetain.DG_REM10_PO1212_aCh3_bWrongParameters	:=	0;
DiagsRetain.DG_REM10_PO1212_aCh4_bOpenSensor	:=	0;
DiagsRetain.DG_REM10_PO1212_aCh4_bOverRange	:=	0;
DiagsRetain.DG_REM10_PO1212_aCh4_bSensorShortCircuit	:=	0;
DiagsRetain.DG_REM10_PO1212_aCh4_bWrongParameters	:=	0;
DiagsRetain.DG_REM10_PO1212_aCh5_bOpenSensor	:=	0;
DiagsRetain.DG_REM10_PO1212_aCh5_bOverRange	:=	0;
DiagsRetain.DG_REM10_PO1212_aCh5_bSensorShortCircuit	:=	0;
DiagsRetain.DG_REM10_PO1212_aCh5_bWrongParameters	:=	0;
DiagsRetain.DG_REM10_PO1212_aCh6_bOpenSensor	:=	0;
DiagsRetain.DG_REM10_PO1212_aCh6_bOverRange	:=	0;
DiagsRetain.DG_REM10_PO1212_aCh6_bSensorShortCircuit	:=	0;
DiagsRetain.DG_REM10_PO1212_aCh6_bWrongParameters	:=	0;
DiagsRetain.DG_REM10_PO1212_aCh7_bOpenSensor	:=	0;
DiagsRetain.DG_REM10_PO1212_aCh7_bOverRange	:=	0;
DiagsRetain.DG_REM10_PO1212_aCh7_bSensorShortCircuit	:=	0;
DiagsRetain.DG_REM10_PO1212_aCh7_bWrongParameters	:=	0;
		
//PO2132		
DiagsRetain.DG_REM10_PO2132_bNoParametrizedModule	:=	0;
DiagsRetain.DG_REM10_PO2132_bPowerSupplyFail	:=	0;
DiagsRetain.DG_REM10_PO2132_aCh0_bOpenSensor	:=	0;
DiagsRetain.DG_REM10_PO2132_aCh0_bWrongParameters	:=	0;
DiagsRetain.DG_REM10_PO2132_aCh1_bOpenSensor	:=	0;
DiagsRetain.DG_REM10_PO2132_aCh1_bWrongParameters	:=	0;
DiagsRetain.DG_REM10_PO2132_aCh2_bOpenSensor	:=	0;
DiagsRetain.DG_REM10_PO2132_aCh2_bWrongParameters	:=	0;
DiagsRetain.DG_REM10_PO2132_aCh3_bOpenSensor	:=	0;
DiagsRetain.DG_REM10_PO2132_aCh3_bWrongParameters	:=	0;

		
//PO9100		
DiagsRetain.DG_REM10_PO9100_bReserved00	:=	0;
		
//PO1000		
DiagsRetain.DG_REM04_PO1000_bHardwareFailure	:=	0;
DiagsRetain.DG_REM04_PO1000_bPowerSupplyFail	:=	0;


// Registra o tempo do sistema
SysTimeGetUs(uliPouEndTime);
// Calcula duração mínima/máxima desta POU
MinMaxTimes.uliPouMinTime_CleanStatus:= MIN(MinMaxTimes.uliPouMinTime_CleanStatus, uliPouEndTime - uliPouIniTime);
MinMaxTimes.uliPouMaxTime_CleanStatus:= MAX(MinMaxTimes.uliPouMaxTime_CleanStatus, uliPouEndTime - uliPouIniTime);

END_PROGRAM

// Device/Application/UserPOUs/ActivePrg
{attribute 'symbol' := 'none'}
PROGRAM ActivePrg
VAR
	ElapsedTime:	TON;		// Temporizador de execução da aplicação
	bStateChangeEnabledByAppl : BOOL := FALSE;
	bRedStatisticsReseted : BOOL := FALSE;
	bStartTimer : BOOL := TRUE;
	uliPouIniTime : ULINT;
	uliPouEndTime : ULINT;
	uliPouAvgTime : ARRAY [1..100] OF ULINT;
	uliPouSumTime : ULINT;
	iPouTimeIndex : INT := 1;
	
	{attribute 'symbol' := 'readwrite'}
	bButton_STBY_PLCA : BOOL; // Comando passar para STANDBY o PLCA
	{attribute 'symbol' := 'readwrite'}
	bButton_INA_PLCA : BOOL; // Comando passar para INATIVO o PLCA
	{attribute 'symbol' := 'readwrite'}
	bButton_STBY_PLCB : BOOL;; // Comando passar para STANDBY o PLCB
	{attribute 'symbol' := 'readwrite'}
	bButton_INA_PLCB : BOOL; // Comando passar para INATIVO o PLCB
	
	uliWantedScanTimeUs:	ULINT;	// Duração desejada para a tarefa apontada na chamada da função [us]
	uliLastCycleDelayUs:	ULINT;			// Atraso realizado nesta chamada, deve realimentar a próxima [us]
	
	
		timeAjust: ULINT; // deletar, investigação
END_VAR

// Registra o tempo do sistema
SysTimeGetUs(uliPouIniTime);

// Atualiza o estado redundante corrente de cada PLC e comandos via supervisório
IF DG_NX4010.tRedundancy.RedDgnLoc.sGeneral_Diag.ePLC_ID = CLUCONF_ID.PLC_A THEN
	PersistentVars.byCurRedStatePlcA:= DG_NX4010.tRedundancy.RedDgnLoc.sGeneral_Diag.eRedState;
	PersistentVars.byCurRedStatePlcB:= DG_NX4010.tRedundancy.RedDgnRem.sGeneral_Diag.eRedState;
	IF bButton_STBY_PLCA THEN DG_NX4010.tRedundancy.RedCmdLoc.bStandbyLocal:= TRUE; bButton_STBY_PLCA:= FALSE; END_IF
	IF bButton_INA_PLCA THEN DG_NX4010.tRedundancy.RedCmdLoc.bInactiveLocal:=TRUE; bButton_INA_PLCA:= FALSE; END_IF
	IF bButton_STBY_PLCB THEN  DG_NX4010.tRedundancy.RedCmdLoc.bStandbyRemote:=TRUE; bButton_STBY_PLCB:= FALSE; END_IF
	IF bButton_INA_PLCB THEN DG_NX4010.tRedundancy.RedCmdLoc.bInactiveRemote:= TRUE; bButton_INA_PLCB:= FALSE; END_IF	
ELSE
	PersistentVars.byCurRedStatePlcA:= DG_NX4010.tRedundancy.RedDgnRem.sGeneral_Diag.eRedState;
	PersistentVars.byCurRedStatePlcB:= DG_NX4010.tRedundancy.RedDgnLoc.sGeneral_Diag.eRedState;
	IF bButton_STBY_PLCB THEN DG_NX4010.tRedundancy.RedCmdLoc.bStandbyLocal:= TRUE; bButton_STBY_PLCB:= FALSE; END_IF
	IF bButton_INA_PLCB THEN DG_NX4010.tRedundancy.RedCmdLoc.bInactiveLocal:=TRUE; bButton_INA_PLCB:= FALSE; END_IF
	IF bButton_STBY_PLCA THEN  DG_NX4010.tRedundancy.RedCmdLoc.bStandbyRemote:=TRUE; bButton_STBY_PLCA:= FALSE; END_IF
	IF bButton_INA_PLCA THEN DG_NX4010.tRedundancy.RedCmdLoc.bInactiveRemote:= TRUE; bButton_INA_PLCA:= FALSE; END_IF	
END_IF

// MODBUS_Server_2: copia o valor das saídas para as entradas
ATs.abyModbus2Status:= ATs.abyModbus2Coils;
ATs.awModbus2InputReg:= ATs.awModbus2Holding;

// MODBUS_Server_3: copia o valor das saídas para as entradas
ATs.abyModbus3Status:= ATs.abyModbus3Coils;
ATs.awModbus3InputReg:= ATs.awModbus3Holding;

// MODBUS_Server_4: copia o valor das saídas para as entradas
ModbusSymbol.abModbus4Status:= ModbusSymbol.abModbus4Coils;
ModbusSymbol.awModbus4InputReg:= ModbusSymbol.awModbus4Holding;


// Função para realizar testes manuais de aumento do tempo de ciclo
uliLastCycleDelayUs:= ForceScanTime('Application', 'MainTask', uliLastCycleDelayUs, uliWantedScanTimeUs);

// Comunicação com o cliente IEC104 da JIGA 11
Iec104Server();

// Retorna se o teste estiver desabilitado
IF Symbolics.bStartTestCopy = FALSE THEN
	RETURN;
END_IF

// Verifica solicitação de reinicialização do super teste
IF Symbolics.bEnableCleanStats_ActivePrg THEN
	// Reinicializa o temporizador de execução
	bStartTimer:= FALSE;
	Symbolics.bEnableCleanStats_CheckProfibusIOs:= TRUE;
	Symbolics.bEnableCleanStats_ActivePrg:= FALSE;
END_IF

// Contabiliza o tempo de teste transcorrido até a ocorrência da falha
IF bStartTimer = FALSE OR PersistentVars.bFailureDetected = FALSE THEN
	ElapsedTime(IN:= bStartTimer, PT:= T#500H, ET=> PersistentVars.tElapsedTimeToFailure);
	bStartTimer:= TRUE;
END_IF

// Se um dos CPs está ativo e o outro reserva...
IF  (DG_NX4010.tRedundancy.RedDgnLoc.sGeneral_Diag.eRedState = REDUNDANCY_STATE.ACTIVE   AND 
     DG_NX4010.tRedundancy.RedDgnRem.sGeneral_Diag.eRedState = REDUNDANCY_STATE.STANDBY) OR
    (DG_NX4010.tRedundancy.RedDgnLoc.sGeneral_Diag.eRedState = REDUNDANCY_STATE.STANDBY  AND 
     DG_NX4010.tRedundancy.RedDgnRem.sGeneral_Diag.eRedState = REDUNDANCY_STATE.ACTIVE)  THEN
	// Habilita a troca de estados de redundância
	bStateChangeEnabledByAppl:= TRUE;
	// Apaga as estatísticas de redundância na primeira vez
	IF bRedStatisticsReseted = FALSE THEN
		DG_NX4010.tRedundancy.RedCmdLoc.bResetNETStatisticsLocal:=  TRUE;
		DG_NX4010.tRedundancy.RedCmdLoc.bResetNETStatisticsRemote:= TRUE;
		bRedStatisticsReseted:= TRUE;
	END_IF
END_IF

IF 	bStateChangeEnabledByAppl = TRUE AND			// Se a troca de estado está habilitada pela aplicação...
	PersistentVars.bEnableStateChange = TRUE AND	// Se a troca de estado está habilitada pelo usuário...
	PersistentVars.bFailureDetected = FALSE AND		// Se ainda não foram identificadas falhas nos testes...
	PersistentVars.bExchangeStateFail = FALSE THEN	// Se ainda não ocorreram falhas de troca de estado...
		// Realiza a troca de estados de redundância
		StateChange();
END_IF

CheckModbus2();			// Consistência dos objetos de comunicação MODBUS Ethernet
CheckModbus3();			// Consistência dos objetos de comunicação MODBUS Ethernet
CheckModbus4();			// Consistência dos objetos de comunicação MODBUS Ethernet

CheckProfibusIOs();		// Consistencia dos módulos de E/S digitais/analógicos Profibus

///CheckRecipe();			// Consitência do Recipe Manager (está comentada devido ao bug 16986, pois gera picos na MainTask)
CheckSoe();				// Consistência do serviço SOE
CheckLanguages();		// Consistência das linguagens de programação

Alarms();				// Detecção dos alarmes mapeados no sistema de supervisão
CheckNVL();				// Consistência do NVL
IncrRedData();			// Incrementa os dados redundantes consistidos pelo PLC reserva
PidGenerator();			// Gera oscilação para testar o PIDControl

// Apenas chama variáveis que estão dentro da GVL
// Não precisa consistir, apenas testar uma GVL grande.
QuantityOfVariables.iTest0000:= QuantityOfVariables.iTest0000 + 1;
QuantityOfVariables.iTest9999:= QuantityOfVariables.iTest0000;
PIDControl();

Recursividade();		// Temporizadores sendo usado em function blocks para pegar problemas de exception na partida (ocorreu na Petrobras)


// Registra o tempo do sistema
SysTimeGetUs(uliPouEndTime);

// Calcula duração média desta POU
uliPouSumTime:= uliPouSumTime - uliPouAvgTime[iPouTimeIndex];
uliPouAvgTime[iPouTimeIndex]:= uliPouEndTime - uliPouIniTime;
uliPouSumTime:= uliPouSumTime + uliPouAvgTime[iPouTimeIndex];
// Calcula duração mínima/média/máxima desta POU
MinMaxTimes.uliPouMinTime_ActivePrg:= MIN(MinMaxTimes.uliPouMinTime_ActivePrg, uliPouAvgTime[iPouTimeIndex]);
MinMaxTimes.uliPouAvgTime_ActivePrg:= uliPouSumTime/(SIZEOF(uliPouAvgTime)/SIZEOF(uliPouAvgTime[1]));
MinMaxTimes.uliPouMaxTime_ActivePrg:= MAX(MinMaxTimes.uliPouMaxTime_ActivePrg, uliPouAvgTime[iPouTimeIndex]);
// Proximo indice para cálculo da duração média desta POU
iPouTimeIndex:= iPouTimeIndex + 1;
IF iPouTimeIndex > ULINT_TO_INT(SIZEOF(uliPouAvgTime)/SIZEOF(uliPouAvgTime[1])) THEN
	iPouTimeIndex:= 1;
END_IF

END_PROGRAM

// ForceScanTime
FUNCTION ForceScanTime : ULINT
VAR_INPUT
	sAppName : STRING;
	sTaskName : STRING;
	uliUsLast : ULINT;
	uliUsWanted : ULINT;
END_VAR
VAR
	uliUsIni : ULINT;
	uliUsNow : ULINT;
	TaskInfo : stTaskInfo;
END_VAR

(*
Função para ajuste da duração de uma tarefa cíclica específica da aplicação:
- deve ser chamada uma única vez e a cada ciclo da tarefa.
- é realimentada: deve ser chamada com o último valor retornado.
- caso retorne zero: a duração da tarefa já é maior que a desejada.
- o jitter é mantido, mas a duração média da tarefa será a desejada.

Exemplo de declaração e chamada para ajuste da duração da tarefa MainTask em 10ms (10.000us):
	
	uliWantedScanTimeUs:	ULINT:= 10000;	// Duração desejada para a tarefa apontada na chamada da função [us]
	uliLastCycleDelayUs:	ULINT;			// Atraso realizado nesta chamada, deve realimentar a próxima [us]
	
	uliLastCycleDelayUs:= ForceScanTime('Application', 'MainTask', uliLastCycleDelayUs, uliWantedScanTimeUs);
*) 

// Registro do tempo inicial
SysTimeCore.SysTimeGetUs(uliUsIni);
// Leitura dos tempos de ciclo da tarefa apontada
NextoStandard.GetTaskInfo(ADR(sAppName), ADR(sTaskName), ADR(TaskInfo));
// Se as estatísticas foram inicializadas...
IF TaskInfo.dwCurScanTime = 0 THEN
	// Vai aguardar a passagem do tempo [us] desejado
	ForceScanTime:= uliUsWanted;
ELSE
	// Calcula novo tempo [us] que deve permanecer em looping
	ForceScanTime:= uliUsLast + uliUsWanted - TaskInfo.dwCurScanTime;
	// Evita exceção por configurar um tempo desejado pequeno demais
	IF ForceScanTime > uliUsWanted THEN ForceScanTime:= 0; END_IF
END_IF
// Permanece em looping até atingir o tempo de ciclo desejado
REPEAT SysTimeCore.SysTimeGetUs(uliUsNow);
UNTIL uliUsNow - uliUsIni > ForceScanTime END_REPEAT

END_FUNCTION

// Device/Application/UserPOUs/Redundant/Iec104Server
PROGRAM Iec104Server
VAR
	diCycleTimeAcc:			DINT;
	diITCounter:			DINT;
	// Variáveis da DbpCmdReceiver
	bDbpCmdSetup:			BOOL:= TRUE;
	byDbpCmdResult:			BYTE;
	fbDbpCmdReceiver:		LibRtuStandard.CommandReceiver;
	// Variáveis da StepCmdReceiver
	bStepCmdSetup:			BOOL:= TRUE;
	byStepCmdResult:		BYTE;
	fbStepCmdReceiver:		LibRtuStandard.CommandReceiver;
	// Variáveis mapeadas no driver IEC104 Server
	bDI:					BOOL;
	bDO:					BOOL;
	dbpI:					LibDataTypes.DBP;
	dbpO:					LibDataTypes.DBP;
	usiSP:					USINT;
	dbpStep:				LibDataTypes.DBP;
	iAIn:					INT;
	iAOn:					INT;
	iAIs:					INT;
	iAOs:					INT;
	rAIf:					REAL;
	rAOf:					REAL;
	diIT:					DINT;
	usiJigId:				USINT:= 3;
END_VAR

// Tratamento dos comandos DBP
Iec104Server.DbpCmdReceiver();
// Tratamento dos comandos Step
Iec104Server.StepCmdReceiver();

// Copia o valor das saídas digitais para as entradas digitais
bDI:= bDO;
dbpI:= dbpO;

// Copia o valor das saídas analógicas para as entradas analógicas
iAIn:= iAOn;
iAIs:= iAOs;
rAIf:= rAOf;

// Acumula o tempo de ciclo
diCycleTimeAcc:= diCycleTimeAcc + ProjectConstants.iMainTaskInterval;
// Incrementa o contador local a cada 100ms
IF diCycleTimeAcc >= 100 THEN
	diCycleTimeAcc:= diCycleTimeAcc - 100;
	diITCounter:= diITCounter + 1;
END_IF

ACTION DbpCmdReceiver:
// Executa a configuração da função no primeiro ciclo
IF bDbpCmdSetup THEN
	bDbpCmdSetup:= FALSE;
	fbDbpCmdReceiver.bExec:= TRUE;
	fbDbpCmdReceiver.dwTimeout:= 256 * 10;
	fbDbpCmdReceiver.eCommandResult:= COMMAND_RESULT.NONE;
END_IF

// Caso um comando seja capturado...
IF fbDbpCmdReceiver.bCommandAvailable THEN
	
	// Trata cada um dos comandos possíveis de serem interceptados
	CASE fbDbpCmdReceiver.sCommand.eCommand OF
		
		COMMAND_TYPE.NO_COMMAND:
			
			// Informar que tem comando disponível mas que não é um comando,
			// é uma situação inválida. Não faz nada. Deve sair por timeout.
			byDbpCmdResult:= 0;
		
		COMMAND_TYPE.SELECT:
			
			// Trata apenas comandos para pontos duplos
			IF fbDbpCmdReceiver.sCommand.sSelectParameters.sValue.eParamType = DOUBLE_POINT_COMMAND THEN
				// Retorna comando finalizado com sucesso (controlado pelo protocolo IEC104)
				byDbpCmdResult:= 7;
			ELSE
				// Retorna comando não suportado
				byDbpCmdResult:= 1;
			END_IF
		
		COMMAND_TYPE.OPERATE:
			
			// Trata apenas comandos para pontos duplos
			IF fbDbpCmdReceiver.sCommand.sOperateParameters.sValue.eParamType = DOUBLE_POINT_COMMAND THEN
				// Geração do pulso nas saídas
				IF fbDbpCmdReceiver.sCommand.sOperateParameters.sValue.sDoublePoint.bValue THEN
					// Executa a função de TRIP
					dbpO.OFF:= FALSE;
					dbpO.ON:= TRUE;
				ELSE
					// Executa a função de CLOSE
					dbpO.OFF:= TRUE;
					dbpO.ON:= FALSE;
				END_IF
				// Retorna comando finalizado com sucesso
				byDbpCmdResult:= 7;
			ELSE
				// Retorna comando não suportado
				byDbpCmdResult:= 1;
			END_IF
		
		COMMAND_TYPE.CANCEL:
			
			// Retorna comando finalizado com sucesso (controlado pelo protocolo IEC104)
			byDbpCmdResult:= 7;
			
	END_CASE
	
	// Trata o resultado da função de comando pulsado
	// e gera a resposta para o comando interceptado
	CASE byDbpCmdResult OF
		1:	// Tipo inválido de comando
			fbDbpCmdReceiver.eCommandResult:= COMMAND_RESULT.NOT_SUPPORTED;
			fbDbpCmdReceiver.bDone:= TRUE;
		2:	// Parâmetros de entrada inválidos
			fbDbpCmdReceiver.eCommandResult:= COMMAND_RESULT.INCONSISTENT_PARAMETERS;
			fbDbpCmdReceiver.bDone:= TRUE;
		3:	// Mudança de parâmetro em execução
			fbDbpCmdReceiver.eCommandResult:= COMMAND_RESULT.PARAMETER_CHANGE_IN_EXECUTION;
			fbDbpCmdReceiver.bDone:= TRUE;
		4:	// Módulo não respondeu ao comando (ausente)
			fbDbpCmdReceiver.eCommandResult:= COMMAND_RESULT.HARDWARE_ERROR;
			fbDbpCmdReceiver.bDone:= TRUE;
		5:	// Comando iniciado e em execução (não retorna nada)
		6:	// Outro comando já foi enviado para este ponto e está em execução
			fbDbpCmdReceiver.eCommandResult:= COMMAND_RESULT.LOCKED_BY_OTHER_CLIENT;
			fbDbpCmdReceiver.bDone:= TRUE;
		7:	// Comando finalizado com sucesso
			fbDbpCmdReceiver.eCommandResult:= COMMAND_RESULT.SUCCESS;
			fbDbpCmdReceiver.bDone:= TRUE;
	END_CASE
	
END_IF

// Inicializa o endereço do comando (ciclicamente, pois é uma UCP redundante)
fbDbpCmdReceiver.dwVariableAddr:= ADR(dbpO);
// Chama o interceptador de comandos
fbDbpCmdReceiver();

IF fbDbpCmdReceiver.bDone THEN
	fbDbpCmdReceiver.bDone:= FALSE;
END_IF
END_ACTION

ACTION StepCmdReceiver:
// Executa a configuração da função no primeiro ciclo
IF bStepCmdSetup THEN
	bStepCmdSetup:= FALSE;
	fbStepCmdReceiver.bExec:= TRUE;
	fbStepCmdReceiver.dwTimeout:= 256 * 10;
	fbStepCmdReceiver.eCommandResult:= COMMAND_RESULT.NONE;
END_IF

// Caso um comando seja capturado...
IF fbStepCmdReceiver.bCommandAvailable THEN
	
	// Trata cada um dos comandos possíveis de serem interceptados
	CASE fbStepCmdReceiver.sCommand.eCommand OF
		
		COMMAND_TYPE.NO_COMMAND:
	
			// Informar que tem comando disponível mas que não é um comando,
			// é uma situação inválida. Não faz nada. Deve sair por timeout.
			byStepCmdResult:= 0;
		
		COMMAND_TYPE.SELECT:
			
			// Trata apenas comandos para pontos duplos
			IF fbStepCmdReceiver.sCommand.sSelectParameters.sValue.eParamType = DOUBLE_POINT_COMMAND THEN
				// Retorna comando finalizado com sucesso (controlado pelo protocolo IEC104)
				byStepCmdResult:= 7;
			ELSE
				// Retorna comando não suportado
				byStepCmdResult:= 1;
			END_IF
		
		COMMAND_TYPE.OPERATE:
			// Trata apenas comandos para pontos duplos
			IF fbStepCmdReceiver.sCommand.sOperateParameters.sValue.eParamType = DOUBLE_POINT_COMMAND THEN
				// Geração do pulso nas saídas
				IF fbStepCmdReceiver.sCommand.sOperateParameters.sValue.sDoublePoint.bValue THEN
					// Executa a função de incremento
					usiSP:= usiSP + 1;
				ELSE
					// Executa a função de decremento
					usiSP:= usiSP - 1;
				END_IF
				// Retorna comando finalizado com sucesso
				byStepCmdResult:= 7;
			ELSE
				// Retorna comando não suportado
				byStepCmdResult:= 1;
			END_IF
		
		COMMAND_TYPE.CANCEL:
			
			// Retorna comando finalizado com sucesso (controlado pelo protocolo IEC104)
			byStepCmdResult:= 7;
			
	END_CASE
	
	// Trata o resultado da função de comando pulsado
	// e gera a resposta para o comando interceptado
	CASE byStepCmdResult OF
		1:	// Tipo inválido de comando
			fbStepCmdReceiver.eCommandResult:= COMMAND_RESULT.NOT_SUPPORTED;
			fbStepCmdReceiver.bDone:= TRUE;
		2:	// Parâmetros de entrada inválidos
			fbStepCmdReceiver.eCommandResult:= COMMAND_RESULT.INCONSISTENT_PARAMETERS;
			fbStepCmdReceiver.bDone:= TRUE;
		3:	// Mudança de parâmetro em execução
			fbStepCmdReceiver.eCommandResult:= COMMAND_RESULT.PARAMETER_CHANGE_IN_EXECUTION;
			fbStepCmdReceiver.bDone:= TRUE;
		4:	// Módulo não respondeu ao comando (ausente)
			fbStepCmdReceiver.eCommandResult:= COMMAND_RESULT.HARDWARE_ERROR;
			fbStepCmdReceiver.bDone:= TRUE;
		5:	// Comando iniciado e em execução (não retorna nada)
		6:	// Outro comando já foi enviado para este ponto e está em execução
			fbStepCmdReceiver.eCommandResult:= COMMAND_RESULT.LOCKED_BY_OTHER_CLIENT;
			fbStepCmdReceiver.bDone:= TRUE;
		7:	// Comando finalizado com sucesso
			fbStepCmdReceiver.eCommandResult:= COMMAND_RESULT.SUCCESS;
			fbStepCmdReceiver.bDone:= TRUE;
	END_CASE
	
END_IF

// Inicializa o endereço do comando (ciclicamente, pois é uma UCP redundante)
fbStepCmdReceiver.dwVariableAddr:= ADR(dbpStep);
// Chama o interceptador de comandos
fbStepCmdReceiver();

IF fbStepCmdReceiver.bDone THEN
	fbStepCmdReceiver.bDone:= FALSE;
END_IF
END_ACTION

END_PROGRAM

// Device/Application/UserPOUs/Redundant/StateChange
PROGRAM StateChange
VAR
	wLowLimit : WORD := 50;
	wHighLimit : WORD := 51; //Alterado de 250 para 51
	wTolerance : WORD := 70;
	byState : BYTE := 1;
	wTime : WORD := 0;
	wTimeout : WORD := 0;
	wLimit : WORD := 50;
	uliPouIniTime : ULINT;
	uliPouEndTime : ULINT;
END_VAR

// Esta POU alterna o estado de redundância dos PLCs automaticamente.
// Ela é chamada pela POU ActivePrg, portanto ela é executada somente pelo CP ativo,
// isto deve ser levado em consideração para compreender o código abaixo.
// Estado inicial: CP A ativo, CP B reserva.

// Registra o tempo do sistema
SysTimeGetUs(uliPouIniTime);

CASE byState OF

	1:	// Aguarda tempo para estabilização da nova UCP ativa
		IF wTime < INT_TO_WORD(ProjectConstants.iTimeToSkipAsActive/ProjectConstants.iMainTaskInterval) THEN
			wTime:= wTime + 1;
		ELSE
			// Indica que concluiu o processo de switch-over
			Symbolics.byStateChangeState:= 1;
			// Próximo estado
			byState:= 2;
		END_IF
	
	2:	// Aguarda wLimit ciclos para a próxima alteração de estados
		IF wTime < wLimit THEN
			wTime:= wTime + 1;
		ELSE
			byState:= 3;
			wTime:= 0;
		END_IF
	
	3: // Manda o CP remoto para INATIVO, CP local permanece em ATIVO
		IF wTimeout > (wLimit + wTolerance) THEN
			PersistentVars.bExchangeStateFail:= TRUE;
		ELSE
			wTimeout:= wTimeout+1;
		END_IF
		IF DG_NX4010.tRedundancy.RedDgnRem.sGeneral_Diag.eRedState = REDUNDANCY_STATE.STANDBY THEN
			PersistentVars.dwTransitionsCnt:= PersistentVars.dwTransitionsCnt+1;
			DG_NX4010.tRedundancy.RedCmdLoc.bInactiveRemote:= TRUE;
			byState:= 4;
			wTimeout:= 0;
		END_IF
	
	4: // Aguarda wLimit ciclos
		IF wTime < wLimit THEN 
			wTime:= wTime + 1;
		ELSE
			byState:= 5;
			wTime:= 0;
		END_IF
	
	5: // Manda o CP remoto para RESERVA, CP local permanece em ATIVO
		IF wTimeout > (wLimit + wTolerance) THEN
			PersistentVars.bExchangeStateFail:= TRUE;
		ELSE
			wTimeout:= wTimeout+1;
		END_IF
		IF DG_NX4010.tRedundancy.RedDgnRem.sGeneral_Diag.eRedState = REDUNDANCY_STATE.INACTIVE THEN 
			PersistentVars.dwTransitionsCnt:= PersistentVars.dwTransitionsCnt + 1;
			DG_NX4010.tRedundancy.RedCmdLoc.bStandbyRemote:= TRUE;
			byState:= 6;
			wTimeout:= 0;
		END_IF
	
	6: // Aguarda wLimit ciclos
		IF wTime < wLimit THEN
			wTime:= wTime + 1;
		ELSE
			byState:= 7;
			wTime:= 0;
		END_IF
		// Verifica se chegou a hora de avisar que um switch-over está próximo de ocorrer
		IF (wLimit - wTime) <= INT_TO_WORD(ProjectConstants.iTimeToWarnBeforeSwitchOver/ProjectConstants.iMainTaskInterval) THEN
			// Indica que em dois segundos irá ocorrer um switch-over
			Symbolics.byStateChangeState:= 2;
		END_IF
	
	7: // Manda o CP remoto para ATIVO e CP local para RESERVA
		IF wTimeout > (wLimit + wTolerance) THEN
			PersistentVars.bExchangeStateFail:= TRUE;
		ELSE
			wTimeout:= wTimeout+1;
		END_IF
		IF DG_NX4010.tRedundancy.RedDgnRem.sGeneral_Diag.eRedState = REDUNDANCY_STATE.STANDBY THEN 
			PersistentVars.dwTransitionsCnt:= PersistentVars.dwTransitionsCnt + 2; // '+2' pois ambos CPs trocaram de estado
			PersistentVars.dwSwitchoverCnt:= PersistentVars.dwSwitchoverCnt + 1;
			DG_NX4010.tRedundancy.RedCmdLoc.bStandbyLocal:= TRUE;
			byState:= 8;
			wTimeout:= 0;
			// Indica que está em processo de switch-over
			Symbolics.byStateChangeState:= 3;
		END_IF
	
	8: 	// Incrementa o valor limite para troca de estados
		wLimit:= wLimit + 1;
		// Mantém a duração de cada estado entre 50 e 250 ciclos
		IF wLimit > wHighLimit THEN
			wLimit:= wLowLimit;
		END_IF
		// Inicia um novo ciclo de troca de estados
		byState:= 1;
	
END_CASE

// Mantém a duração de cada estado entre 50 e 250 ciclos

// Registra o tempo do sistema
SysTimeGetUs(uliPouEndTime);
// Calcula duração mínima/máxima desta POU
MinMaxTimes.uliPouMinTime_StateChange:= MIN(MinMaxTimes.uliPouMinTime_StateChange, uliPouEndTime - uliPouIniTime);
MinMaxTimes.uliPouMaxTime_StateChange:= MAX(MinMaxTimes.uliPouMaxTime_StateChange, uliPouEndTime - uliPouIniTime);

END_PROGRAM

// Device/Application/UserPOUs/Non-Redundant/CheckModbus2
PROGRAM CheckModbus2
VAR
	byIndex : BYTE;
	wIndex : WORD;
	bStatusCoil : BOOL;
	bStatusStatus : BOOL;
	bStatusHolding : BOOL;
	bStatusInputReg : BOOL;
	liDigitalTimer : LINT := 0;
	liAnalogTimer : LINT := 0;
	abyCoilsError_DataWr : ARRAY [0..119] OF BYTE;
	abyCoilsError_DataRd : ARRAY [0..119] OF BYTE;
	abyStatusError_DataWr : ARRAY [0..119] OF BYTE;
	abyStatusError_DataRd : ARRAY [0..119] OF BYTE;
	awHoldingError_DataWr : ARRAY [0..119] OF WORD;
	awHoldingError_DataRd : ARRAY [0..119] OF WORD;
	awInputRegError_DataWr : ARRAY [0..119] OF WORD;
	awInputRegError_DataRd : ARRAY [0..119] OF WORD;
	wOldRXNormalResponses : WORD;
	iMilisecondsCounter : INT;
	iBytesPerResponse : INT := 240;
	uliPouIniTime : ULINT;
	uliPouEndTime : ULINT;
END_VAR

// Consistencia da integridade dos dados trocados via MODBUS

// Registra o tempo do sistema
SysTimeGetUs(uliPouIniTime);

//
// Controle e consistência dos coils e input status
//

// Consiste os valores lidos
bStatusCoil:= TRUE;
bStatusStatus:= TRUE;
FOR byIndex:= 0 TO 119 BY 1 DO
	bStatusCoil:= bStatusCoil AND (ATs.abyModbus2CoilsRead[byIndex] = ATs.abyModbus2CoilsWrite[byIndex]);
	bStatusStatus:= bStatusStatus AND (ATs.abyModbus2StatusRead[byIndex] = ATs.abyModbus2CoilsWrite[byIndex]);
END_FOR

// Se o estado de redundância deste PLC alterou...
IF NonRedData.bRedStateChanged THEN
	// Torna as saídas diferentes das entradas, garantindo que as consistências de dados
	// sejam feitas a partir de valores decorrentes de novas comunicações
	ATs.abyModbus2CoilsWrite[0]:= ATs.abyModbus2StatusRead[0] + 10;
	// Inicializa temporizador para atrasar a consistência dos valores lidos, pois quando
	// o PLC assume como ativo, vai levar algum tempo até a comunicação ser estabelecida
	liDigitalTimer:= - ProjectConstants.iTimeToSkipAsActive;
ELSE
	// Se o protocolo MODBUS está rodando e se os dados são consistentes...
	IF DG_MODBUS_Client_2.tDiag.bRunning AND bStatusCoil AND bStatusStatus THEN
		// Altera o valor a ser escrito nos coils
		ATs.abyModbus2CoilsWrite[0]:= ATs.abyModbus2CoilsWrite[0] + 10;
		// Reseta o temporizador
		liDigitalTimer:= 0;
	ELSE
		// Acumula o tempo que passou
		liDigitalTimer:= liDigitalTimer + ProjectConstants.iMainTaskInterval;
		// Registra o tempo máximo
		MinMaxTimes.liDigMaxTime_CheckModbus2:= MAX(MinMaxTimes.liDigMaxTime_CheckModbus2, liDigitalTimer);
		// Caso o tempo máximo tenha sido extrapolado...
		IF liDigitalTimer >= ProjectConstants.iModbus2ReadWriteDelay THEN
			// Registra falha nos coils, caso tenha ocorrido
			IF bStatusCoil = FALSE THEN
				PersistentVars.bModbus2ErrorCoil:= TRUE;
				abyCoilsError_DataWr:= ATs.abyModbus2CoilsWrite;
				abyCoilsError_DataRd:= ATs.abyModbus2CoilsRead;
			END_IF
			// Registra falha nos inputs, caso tenha ocorrido
			IF bStatusStatus = FALSE THEN
				PersistentVars.bModbus2ErrorStatus:= TRUE;
				abyStatusError_DataWr:= ATs.abyModbus2CoilsWrite;
				abyStatusError_DataRd:= ATs.abyModbus2StatusRead;
			END_IF
		END_IF
	END_IF
END_IF

// Atualiza os valores escritos
FOR byIndex:= 1 TO 119 BY 1 DO
	ATs.abyModbus2CoilsWrite[byIndex]:= ATs.abyModbus2CoilsWrite[byIndex - 1] + byIndex;
END_FOR

//
// Controle e consistência dos holding e input registers
//

// Consiste os valores lidos
bStatusHolding:= TRUE;
bStatusInputReg:= TRUE;
FOR wIndex:= 0 TO 119 BY 1 DO
	bStatusHolding:= bStatusHolding AND (ATs.awModbus2HoldingRead[wIndex] = ATs.awModbus2HoldingWrite[wIndex]);
	bStatusInputReg:= bStatusInputReg AND (ATs.awModbus2InputRegRead[wIndex] = ATs.awModbus2HoldingWrite[wIndex]);
END_FOR

// Se o estado de redundância deste PLC alterou...
IF NonRedData.bRedStateChanged THEN
	// Torna as saídas diferentes das entradas, garantindo que as consistências de dados
	// sejam feitas a partir de valores decorrentes de novas comunicações
	ATs.awModbus2HoldingWrite[0]:= ATs.awModbus2InputRegRead[0] + 100;
	// Inicializa temporizador para atrasar a consistência dos valores lidos, pois quando
	// o PLC assume como ativo, vai levar algum tempo até a comunicação ser estabelecida
	liAnalogTimer:= - ProjectConstants.iTimeToSkipAsActive;
ELSE
	// Se o protocolo MODBUS está rodando e se os dados são consistentes...
	IF DG_MODBUS_Client_2.tDiag.bRunning AND bStatusHolding AND bStatusInputReg THEN
		// Incrementa o valor escrito nos holding registers
		ATs.awModbus2HoldingWrite[0]:= ATs.awModbus2HoldingWrite[0] + 100;
		// Reseta o temporizador
		liAnalogTimer:= 0;
	ELSE
		// Acumula o tempo que passou
		liAnalogTimer:= liAnalogTimer + ProjectConstants.iMainTaskInterval;
		// Registra o tempo máximo
		MinMaxTimes.liAnaMaxTime_CheckModbus2:= MAX(MinMaxTimes.liAnaMaxTime_CheckModbus2, liAnalogTimer);
		// Caso o tempo máximo tenha sido extrapolado...
		IF liAnalogTimer >= ProjectConstants.iModbus2ReadWriteDelay THEN
			// Registra falha nos holding register, caso tenha ocorrido
			IF bStatusHolding = FALSE THEN
				PersistentVars.bModbus2ErrorHolding:= TRUE;
				awHoldingError_DataWr:= ATs.awModbus2HoldingWrite;
				awHoldingError_DataRd:= ATs.awModbus2HoldingRead;
			END_IF
			// Registra falha nos input register, caso tenha ocorrido
			IF bStatusInputReg = FALSE THEN
				PersistentVars.bModbus2ErrorInputReg:= TRUE;
				awInputRegError_DataWr:= ATs.awModbus2HoldingWrite;
				awInputRegError_DataRd:= ATs.awModbus2InputRegRead;
			END_IF
		END_IF
	END_IF
END_IF

// Atualiza os valores escritos
FOR wIndex:= 1 TO 119 BY 1 DO
	ATs.awModbus2HoldingWrite[wIndex]:= ATs.awModbus2HoldingWrite[wIndex - 1] + wIndex;
END_FOR

//
// Calcula a taxa média de comunicação
//

// Incrementa o número de milisegundos que transcorreram
iMilisecondsCounter:= iMilisecondsCounter + ProjectConstants.iMainTaskInterval;
// Se já se passou o tempo configurado desde a última média realizada...
IF iMilisecondsCounter >= ProjectConstants.iMsToComputeComRate THEN
	// Só calcula se o contador não virou
	IF DG_MODBUS_Client_2.tStat.wRXNormalResponses > wOldRXNormalResponses THEN
		// Calcula a taxa de comunicação atual
		MinMaxTimes.diModbus2BytesPerSec:=	WORD_TO_DINT(DG_MODBUS_Client_2.tStat.wRXNormalResponses - wOldRXNormalResponses) *
											iBytesPerResponse * 1000 / iMilisecondsCounter;
	END_IF
	// Zera o número de milisegundos transcorridos
	iMilisecondsCounter:= 0;
	// Salva número de respostas atuais
	wOldRXNormalResponses:= DG_MODBUS_Client_2.tStat.wRXNormalResponses;
END_IF

// Registra o tempo do sistema
SysTimeGetUs(uliPouEndTime);
// Calcula duração mínima/máxima desta POU
MinMaxTimes.uliPouMinTime_CheckModbus2:= MIN(MinMaxTimes.uliPouMinTime_CheckModbus2, uliPouEndTime - uliPouIniTime);
MinMaxTimes.uliPouMaxTime_CheckModbus2:= MAX(MinMaxTimes.uliPouMaxTime_CheckModbus2, uliPouEndTime - uliPouIniTime);

END_PROGRAM

// Device/Application/UserPOUs/Non-Redundant/CheckModbus3
PROGRAM CheckModbus3
VAR
	byIndex : BYTE;
	wIndex : WORD;
	bStatusCoil : BOOL;
	bStatusStatus : BOOL;
	bStatusHolding : BOOL;
	bStatusInputReg : BOOL;
	liDigitalTimer : LINT := 0;
	liAnalogTimer : LINT := 0;
	abyCoilsError_DataWr : ARRAY [0..119] OF BYTE;
	abyCoilsError_DataRd : ARRAY [0..119] OF BYTE;
	abyStatusError_DataWr : ARRAY [0..119] OF BYTE;
	abyStatusError_DataRd : ARRAY [0..119] OF BYTE;
	awHoldingError_DataWr : ARRAY [0..119] OF WORD;
	awHoldingError_DataRd : ARRAY [0..119] OF WORD;
	awInputRegError_DataWr : ARRAY [0..119] OF WORD;
	awInputRegError_DataRd : ARRAY [0..119] OF WORD;
	wOldRXNormalResponses : WORD;
	iMilisecondsCounter : INT;
	iBytesPerResponse : INT := 240;
	uliPouIniTime : ULINT;
	uliPouEndTime : ULINT;
END_VAR

// Consistencia da integridade dos dados trocados via MODBUS

// Registra o tempo do sistema
SysTimeGetUs(uliPouIniTime);

//
// Controle e consistência dos coils e input status
//

// Consiste os valores lidos
bStatusCoil:= TRUE;
bStatusStatus:= TRUE;
FOR byIndex:= 0 TO 119 BY 1 DO
	bStatusCoil:= bStatusCoil AND (ATs.abyModbus3CoilsRead[byIndex] = ATs.abyModbus3CoilsWrite[byIndex]);
	bStatusStatus:= bStatusStatus AND (ATs.abyModbus3StatusRead[byIndex] = ATs.abyModbus3CoilsWrite[byIndex]);
END_FOR

// Se o estado de redundância deste PLC alterou...
IF NonRedData.bRedStateChanged THEN
	// Torna as saídas diferentes das entradas, garantindo que as consistências de dados
	// sejam feitas a partir de valores decorrentes de novas comunicações
	ATs.abyModbus3CoilsWrite[0]:= ATs.abyModbus3StatusRead[0] + 10;
	// Inicializa temporizador para atrasar a consistência dos valores lidos, pois quando
	// o PLC assume como ativo, vai levar algum tempo até a comunicação ser estabelecida
	liDigitalTimer:= - ProjectConstants.iTimeToSkipAsActive;
ELSE
	// Se o protocolo MODBUS está rodando e se os dados são consistentes...
	IF DG_MODBUS_Client_3.tDiag.bRunning AND bStatusCoil AND bStatusStatus THEN
		// Altera o valor a ser escrito nos coils
		ATs.abyModbus3CoilsWrite[0]:= ATs.abyModbus3CoilsWrite[0] + 10;
		// Reseta o temporizador
		liDigitalTimer:= 0;
	ELSE
		// Acumula o tempo que passou
		liDigitalTimer:= liDigitalTimer + ProjectConstants.iMainTaskInterval;
		// Registra o tempo máximo
		MinMaxTimes.liDigMaxTime_CheckModbus3:= MAX(MinMaxTimes.liDigMaxTime_CheckModbus3, liDigitalTimer);
		// Caso o tempo máximo tenha sido extrapolado...
		IF liDigitalTimer >= ProjectConstants.iModbus3ReadWriteDelay THEN
			// Restarta o MODBUS caso o bug 17184 se manifeste.
			IF DG_MODBUS_Server_3.tStat.wActiveConnections = 0 THEN
				///DG_MODBUS_Server_3.tCommand.bRestart:= TRUE;
				PersistentVars.iBug17184_CounterDig_MDBUS3:= PersistentVars.iBug17184_CounterDig_MDBUS3 + 1;
				///iDigitalTimer:= - ProjectConstants.iTimeToSkipAsActive;
			ELSE	
				// Registra falha nos coils, caso tenha ocorrido
				IF bStatusCoil = FALSE THEN
					PersistentVars.bModbus3ErrorCoil:= TRUE;
					abyCoilsError_DataWr:= ATs.abyModbus3CoilsWrite;
					abyCoilsError_DataRd:= ATs.abyModbus3CoilsRead;
				END_IF
				// Registra falha nos inputs, caso tenha ocorrido
				IF bStatusStatus = FALSE THEN
					PersistentVars.bModbus3ErrorStatus:= TRUE;
					abyStatusError_DataWr:= ATs.abyModbus3CoilsWrite;
					abyStatusError_DataRd:= ATs.abyModbus3StatusRead;
				END_IF
			END_IF
		END_IF
	END_IF
END_IF

// Atualiza os valores escritos
FOR byIndex:= 1 TO 119 BY 1 DO
	ATs.abyModbus3CoilsWrite[byIndex]:= ATs.abyModbus3CoilsWrite[byIndex - 1] + byIndex;
END_FOR

//
// Controle e consistência dos holding e input registers
//

// Consiste os valores lidos
bStatusHolding:= TRUE;
bStatusInputReg:= TRUE;
FOR wIndex:= 0 TO 119 BY 1 DO
	bStatusHolding:= bStatusHolding AND (ATs.awModbus3HoldingRead[wIndex] = ATs.awModbus3HoldingWrite[wIndex]);
	bStatusInputReg:= bStatusInputReg AND (ATs.awModbus3InputRegRead[wIndex] = ATs.awModbus3HoldingWrite[wIndex]);
END_FOR

